# B&R Automation Studio project AAU12Segmenter (part 2)

```iecst
	::OutputVariables[1,0]	AT %QB."KUKA2_KRC4_ProfiNet_5_0".Module001_8_digital_outputs_O_00;
	::OutputVariables[1,1]	AT %QB."KUKA2_KRC4_ProfiNet_5_0".Module001_8_digital_outputs_O_01;
	::OutputVariables[1,2]	AT %QB."KUKA2_KRC4_ProfiNet_5_0".Module001_8_digital_outputs_O_02;
	::OutputVariables[1,3]	AT %QB."KUKA2_KRC4_ProfiNet_5_0".Module001_8_digital_outputs_O_03;
	::OutputVariables[1,4]	AT %QB."KUKA2_KRC4_ProfiNet_5_0".Module001_8_digital_outputs_O_04;
	::OutputVariables[1,5]	AT %QB."KUKA2_KRC4_ProfiNet_5_0".Module001_8_digital_outputs_O_05;
	::OutputVariables[1,6]	AT %QB."KUKA2_KRC4_ProfiNet_5_0".Module001_8_digital_outputs_O_06;
	::OutputVariables[1,7]	AT %QB."KUKA2_KRC4_ProfiNet_5_0".Module001_8_digital_outputs_O_07;
	::OutputVariables[1,8]	AT %QB."KUKA2_KRC4_ProfiNet_5_0".Module001_8_digital_outputs_O_08;
	::OutputVariables[1,9]	AT %QB."KUKA2_KRC4_ProfiNet_5_0".Module001_8_digital_outputs_O_09;
	::OutputVariables[1,10]	AT %QB."KUKA2_KRC4_ProfiNet_5_0".Module001_8_digital_outputs_O_10;
	::OutputVariables[1,11]	AT %QB."KUKA2_KRC4_ProfiNet_5_0".Module001_8_digital_outputs_O_11;
	::OutputVariables[1,12]	AT %QB."KUKA2_KRC4_ProfiNet_5_0".Module001_8_digital_outputs_O_12;
	::OutputVariables[1,13]	AT %QB."KUKA2_KRC4_ProfiNet_5_0".Module001_8_digital_outputs_O_13;
	::OutputVariables[1,14]	AT %QB."KUKA2_KRC4_ProfiNet_5_0".Module001_8_digital_outputs_O_14;
	::OutputVariables[1,15]	AT %QB."KUKA2_KRC4_ProfiNet_5_0".Module001_8_digital_outputs_O_15;
	::OutputVariables[1,16]	AT %QB."KUKA2_KRC4_ProfiNet_5_0".Module001_8_digital_outputs_O_16;
	::OutputVariables[1,17]	AT %QB."KUKA2_KRC4_ProfiNet_5_0".Module001_8_digital_outputs_O_17;
	::OutputVariables[1,18]	AT %QB."KUKA2_KRC4_ProfiNet_5_0".Module001_8_digital_outputs_O_18;
	::OutputVariables[1,19]	AT %QB."KUKA2_KRC4_ProfiNet_5_0".Module001_8_digital_outputs_O_19;
	::OutputVariables[1,20]	AT %QB."KUKA2_KRC4_ProfiNet_5_0".Module001_8_digital_outputs_O_20;
	::OutputVariables[1,21]	AT %QB."KUKA2_KRC4_ProfiNet_5_0".Module001_8_digital_outputs_O_21;
	::OutputVariables[1,22]	AT %QB."KUKA2_KRC4_ProfiNet_5_0".Module001_8_digital_outputs_O_22;
	::OutputVariables[1,23]	AT %QB."KUKA2_KRC4_ProfiNet_5_0".Module001_8_digital_outputs_O_23;
	::OutputVariables[1,24]	AT %QB."KUKA2_KRC4_ProfiNet_5_0".Module001_8_digital_outputs_O_24;
	::OutputVariables[1,25]	AT %QB."KUKA2_KRC4_ProfiNet_5_0".Module001_8_digital_outputs_O_25;
	::OutputVariables[1,26]	AT %QB."KUKA2_KRC4_ProfiNet_5_0".Module001_8_digital_outputs_O_26;
	::OutputVariables[1,27]	AT %QB."KUKA2_KRC4_ProfiNet_5_0".Module001_8_digital_outputs_O_27;
	::OutputVariables[1,28]	AT %QB."KUKA2_KRC4_ProfiNet_5_0".Module001_8_digital_outputs_O_28;
	::OutputVariables[1,29]	AT %QB."KUKA2_KRC4_ProfiNet_5_0".Module001_8_digital_outputs_O_29;
	::OutputVariables[1,30]	AT %QB."KUKA2_KRC4_ProfiNet_5_0".Module001_8_digital_outputs_O_30;
	::OutputVariables[1,31]	AT %QB."KUKA2_KRC4_ProfiNet_5_0".Module001_8_digital_outputs_O_31;
	::OutputVariables[1,32]	AT %QB."KUKA2_KRC4_ProfiNet_5_0".Module001_8_digital_outputs_O_32;
	::OutputVariables[1,33]	AT %QB."KUKA2_KRC4_ProfiNet_5_0".Module001_8_digital_outputs_O_33;
	::OutputVariables[1,34]	AT %QB."KUKA2_KRC4_ProfiNet_5_0".Module001_8_digital_outputs_O_34;
	::OutputVariables[1,35]	AT %QB."KUKA2_KRC4_ProfiNet_5_0".Module001_8_digital_outputs_O_35;
	::OutputVariables[1,36]	AT %QB."KUKA2_KRC4_ProfiNet_5_0".Module001_8_digital_outputs_O_36;
	::OutputVariables[1,37]	AT %QB."KUKA2_KRC4_ProfiNet_5_0".Module001_8_digital_outputs_O_37;
	::OutputVariables[1,38]	AT %QB."KUKA2_KRC4_ProfiNet_5_0".Module001_8_digital_outputs_O_38;
	::OutputVariables[1,39]	AT %QB."KUKA2_KRC4_ProfiNet_5_0".Module001_8_digital_outputs_O_39;
	::OutputVariables[1,40]	AT %QB."KUKA2_KRC4_ProfiNet_5_0".Module001_8_digital_outputs_O_40;
	::OutputVariables[1,41]	AT %QB."KUKA2_KRC4_ProfiNet_5_0".Module001_8_digital_outputs_O_41;
	::OutputVariables[1,42]	AT %QB."KUKA2_KRC4_ProfiNet_5_0".Module001_8_digital_outputs_O_42;
	::OutputVariables[1,43]	AT %QB."KUKA2_KRC4_ProfiNet_5_0".Module001_8_digital_outputs_O_43;
	::OutputVariables[1,44]	AT %QB."KUKA2_KRC4_ProfiNet_5_0".Module001_8_digital_outputs_O_44;
	::OutputVariables[1,45]	AT %QB."KUKA2_KRC4_ProfiNet_5_0".Module001_8_digital_outputs_O_45;
	::OutputVariables[1,46]	AT %QB."KUKA2_KRC4_ProfiNet_5_0".Module001_8_digital_outputs_O_46;
	::OutputVariables[1,47]	AT %QB."KUKA2_KRC4_ProfiNet_5_0".Module001_8_digital_outputs_O_47;
	::OutputVariables[1,48]	AT %QB."KUKA2_KRC4_ProfiNet_5_0".Module001_8_digital_outputs_O_48;
	::OutputVariables[1,49]	AT %QB."KUKA2_KRC4_ProfiNet_5_0".Module001_8_digital_outputs_O_49;
	::OutputVariables[1,50]	AT %QB."KUKA2_KRC4_ProfiNet_5_0".Module001_8_digital_outputs_O_50;
	::OutputVariables[1,51]	AT %QB."KUKA2_KRC4_ProfiNet_5_0".Module001_8_digital_outputs_O_51;
	::OutputVariables[1,52]	AT %QB."KUKA2_KRC4_ProfiNet_5_0".Module001_8_digital_outputs_O_52;
	::OutputVariables[1,53]	AT %QB."KUKA2_KRC4_ProfiNet_5_0".Module001_8_digital_outputs_O_53;
	::OutputVariables[1,54]	AT %QB."KUKA2_KRC4_ProfiNet_5_0".Module001_8_digital_outputs_O_54;
	::OutputVariables[1,55]	AT %QB."KUKA2_KRC4_ProfiNet_5_0".Module001_8_digital_outputs_O_55;
	::OutputVariables[1,56]	AT %QB."KUKA2_KRC4_ProfiNet_5_0".Module001_8_digital_outputs_O_56;
	::OutputVariables[1,57]	AT %QB."KUKA2_KRC4_ProfiNet_5_0".Module001_8_digital_outputs_O_57;
	::OutputVariables[1,58]	AT %QB."KUKA2_KRC4_ProfiNet_5_0".Module001_8_digital_outputs_O_58;
	::OutputVariables[1,59]	AT %QB."KUKA2_KRC4_ProfiNet_5_0".Module001_8_digital_outputs_O_59;
	::OutputVariables[1,60]	AT %QB."KUKA2_KRC4_ProfiNet_5_0".Module001_8_digital_outputs_O_60;
	::OutputVariables[1,61]	AT %QB."KUKA2_KRC4_ProfiNet_5_0".Module001_8_digital_outputs_O_61;
	::OutputVariables[1,62]	AT %QB."KUKA2_KRC4_ProfiNet_5_0".Module001_8_digital_outputs_O_62;
	::OutputVariables[1,63]	AT %QB."KUKA2_KRC4_ProfiNet_5_0".Module001_8_digital_outputs_O_63;
	::OutputVariables[1,64]	AT %QB."KUKA2_KRC4_ProfiNet_5_0".Module001_8_digital_outputs_O_64;
	::OutputVariables[1,65]	AT %QB."KUKA2_KRC4_ProfiNet_5_0".Module001_8_digital_outputs_O_65;
	::OutputVariables[1,66]	AT %QB."KUKA2_KRC4_ProfiNet_5_0".Module001_8_digital_outputs_O_66;
	::OutputVariables[1,67]	AT %QB."KUKA2_KRC4_ProfiNet_5_0".Module001_8_digital_outputs_O_67;
	::OutputVariables[1,68]	AT %QB."KUKA2_KRC4_ProfiNet_5_0".Module001_8_digital_outputs_O_68;
	::OutputVariables[1,69]	AT %QB."KUKA2_KRC4_ProfiNet_5_0".Module001_8_digital_outputs_O_69;
	::OutputVariables[1,70]	AT %QB."KUKA2_KRC4_ProfiNet_5_0".Module001_8_digital_outputs_O_70;
	::OutputVariables[1,71]	AT %QB."KUKA2_KRC4_ProfiNet_5_0".Module001_8_digital_outputs_O_71;
	::OutputVariables[1,72]	AT %QB."KUKA2_KRC4_ProfiNet_5_0".Module001_8_digital_outputs_O_72;
	::OutputVariables[1,73]	AT %QB."KUKA2_KRC4_ProfiNet_5_0".Module001_8_digital_outputs_O_73;
	::OutputVariables[1,74]	AT %QB."KUKA2_KRC4_ProfiNet_5_0".Module001_8_digital_outputs_O_74;
	::OutputVariables[1,75]	AT %QB."KUKA2_KRC4_ProfiNet_5_0".Module001_8_digital_outputs_O_75;
	::OutputVariables[1,76]	AT %QB."KUKA2_KRC4_ProfiNet_5_0".Module001_8_digital_outputs_O_76;
	::OutputVariables[1,77]	AT %QB."KUKA2_KRC4_ProfiNet_5_0".Module001_8_digital_outputs_O_77;
	::OutputVariables[1,78]	AT %QB."KUKA2_KRC4_ProfiNet_5_0".Module001_8_digital_outputs_O_78;
	::OutputVariables[1,79]	AT %QB."KUKA2_KRC4_ProfiNet_5_0".Module001_8_digital_outputs_O_79;
	::OutputVariables[1,80]	AT %QB."KUKA2_KRC4_ProfiNet_5_0".Module001_8_digital_outputs_O_80;
	::OutputVariables[1,81]	AT %QB."KUKA2_KRC4_ProfiNet_5_0".Module001_8_digital_outputs_O_81;
	::OutputVariables[1,82]	AT %QB."KUKA2_KRC4_ProfiNet_5_0".Module001_8_digital_outputs_O_82;
	::OutputVariables[1,83]	AT %QB."KUKA2_KRC4_ProfiNet_5_0".Module001_8_digital_outputs_O_83;
	::OutputVariables[1,84]	AT %QB."KUKA2_KRC4_ProfiNet_5_0".Module001_8_digital_outputs_O_84;
	::OutputVariables[1,85]	AT %QB."KUKA2_KRC4_ProfiNet_5_0".Module001_8_digital_outputs_O_85;
	::OutputVariables[1,86]	AT %QB."KUKA2_KRC4_ProfiNet_5_0".Module001_8_digital_outputs_O_86;
	::OutputVariables[1,87]	AT %QB."KUKA2_KRC4_ProfiNet_5_0".Module001_8_digital_outputs_O_87;
	::OutputVariables[1,88]	AT %QB."KUKA2_KRC4_ProfiNet_5_0".Module001_8_digital_outputs_O_88;
	::OutputVariables[1,89]	AT %QB."KUKA2_KRC4_ProfiNet_5_0".Module001_8_digital_outputs_O_89;
	::OutputVariables[1,90]	AT %QB."KUKA2_KRC4_ProfiNet_5_0".Module001_8_digital_outputs_O_90;
	::OutputVariables[1,91]	AT %QB."KUKA2_KRC4_ProfiNet_5_0".Module001_8_digital_outputs_O_91;
	::OutputVariables[1,92]	AT %QB."KUKA2_KRC4_ProfiNet_5_0".Module001_8_digital_outputs_O_92;
	::OutputVariables[1,93]	AT %QB."KUKA2_KRC4_ProfiNet_5_0".Module001_8_digital_outputs_O_93;
	::OutputVariables[1,94]	AT %QB."KUKA2_KRC4_ProfiNet_5_0".Module001_8_digital_outputs_O_94;
	::OutputVariables[1,95]	AT %QB."KUKA2_KRC4_ProfiNet_5_0".Module001_8_digital_outputs_O_95;
	::OutputVariables[1,96]	AT %QB."KUKA2_KRC4_ProfiNet_5_0".Module001_8_digital_outputs_O_96;
	::OutputVariables[1,97]	AT %QB."KUKA2_KRC4_ProfiNet_5_0".Module001_8_digital_outputs_O_97;
	::OutputVariables[1,98]	AT %QB."KUKA2_KRC4_ProfiNet_5_0".Module001_8_digital_outputs_O_98;
	::OutputVariables[1,99]	AT %QB."KUKA2_KRC4_ProfiNet_5_0".Module001_8_digital_outputs_O_99;
	::OutputVariables[1,100]	AT %QB."KUKA2_KRC4_ProfiNet_5_0".Module001_8_digital_outputs_O_100;
	::OutputVariables[1,101]	AT %QB."KUKA2_KRC4_ProfiNet_5_0".Module001_8_digital_outputs_O_101;
	::OutputVariables[1,102]	AT %QB."KUKA2_KRC4_ProfiNet_5_0".Module001_8_digital_outputs_O_102;
	::OutputVariables[1,103]	AT %QB."KUKA2_KRC4_ProfiNet_5_0".Module001_8_digital_outputs_O_103;
	::OutputVariables[1,104]	AT %QB."KUKA2_KRC4_ProfiNet_5_0".Module001_8_digital_outputs_O_104;
	::OutputVariables[1,105]	AT %QB."KUKA2_KRC4_ProfiNet_5_0".Module001_8_digital_outputs_O_105;
	::OutputVariables[1,106]	AT %QB."KUKA2_KRC4_ProfiNet_5_0".Module001_8_digital_outputs_O_106;
	::OutputVariables[1,107]	AT %QB."KUKA2_KRC4_ProfiNet_5_0".Module001_8_digital_outputs_O_107;
	::OutputVariables[1,108]	AT %QB."KUKA2_KRC4_ProfiNet_5_0".Module001_8_digital_outputs_O_108;
	::OutputVariables[1,109]	AT %QB."KUKA2_KRC4_ProfiNet_5_0".Module001_8_digital_outputs_O_109;
	::OutputVariables[1,110]	AT %QB."KUKA2_KRC4_ProfiNet_5_0".Module001_8_digital_outputs_O_110;
	::OutputVariables[1,111]	AT %QB."KUKA2_KRC4_ProfiNet_5_0".Module001_8_digital_outputs_O_111;
	::OutputVariables[1,112]	AT %QB."KUKA2_KRC4_ProfiNet_5_0".Module001_8_digital_outputs_O_112;
	::OutputVariables[1,113]	AT %QB."KUKA2_KRC4_ProfiNet_5_0".Module001_8_digital_outputs_O_113;
	::OutputVariables[1,114]	AT %QB."KUKA2_KRC4_ProfiNet_5_0".Module001_8_digital_outputs_O_114;
	::OutputVariables[1,115]	AT %QB."KUKA2_KRC4_ProfiNet_5_0".Module001_8_digital_outputs_O_115;
	::OutputVariables[1,116]	AT %QB."KUKA2_KRC4_ProfiNet_5_0".Module001_8_digital_outputs_O_116;
	::OutputVariables[1,117]	AT %QB."KUKA2_KRC4_ProfiNet_5_0".Module001_8_digital_outputs_O_117;
	::OutputVariables[1,118]	AT %QB."KUKA2_KRC4_ProfiNet_5_0".Module001_8_digital_outputs_O_118;
	::OutputVariables[1,119]	AT %QB."KUKA2_KRC4_ProfiNet_5_0".Module001_8_digital_outputs_O_119;
	::OutputVariables[1,120]	AT %QB."KUKA2_KRC4_ProfiNet_5_0".Module001_8_digital_outputs_O_120;
	::OutputVariables[1,121]	AT %QB."KUKA2_KRC4_ProfiNet_5_0".Module001_8_digital_outputs_O_121;
	::OutputVariables[1,122]	AT %QB."KUKA2_KRC4_ProfiNet_5_0".Module001_8_digital_outputs_O_122;
	::OutputVariables[1,123]	AT %QB."KUKA2_KRC4_ProfiNet_5_0".Module001_8_digital_outputs_O_123;
	::OutputVariables[1,124]	AT %QB."KUKA2_KRC4_ProfiNet_5_0".Module001_8_digital_outputs_O_124;
	::OutputVariables[1,125]	AT %QB."KUKA2_KRC4_ProfiNet_5_0".Module001_8_digital_outputs_O_125;
	::OutputVariables[1,126]	AT %QB."KUKA2_KRC4_ProfiNet_5_0".Module001_8_digital_outputs_O_126;
	::OutputVariables[1,127]	AT %QB."KUKA2_KRC4_ProfiNet_5_0".Module001_8_digital_outputs_O_127;
	::OutputVariables[1,128]	AT %QB."KUKA2_KRC4_ProfiNet_5_0".Module001_8_digital_outputs_O_128;
	::OutputVariables[1,129]	AT %QB."KUKA2_KRC4_ProfiNet_5_0".Module001_8_digital_outputs_O_129;
	::OutputVariables[1,130]	AT %QB."KUKA2_KRC4_ProfiNet_5_0".Module001_8_digital_outputs_O_130;
	::OutputVariables[1,131]	AT %QB."KUKA2_KRC4_ProfiNet_5_0".Module001_8_digital_outputs_O_131;
	::OutputVariables[1,132]	AT %QB."KUKA2_KRC4_ProfiNet_5_0".Module001_8_digital_outputs_O_132;
	::OutputVariables[1,133]	AT %QB."KUKA2_KRC4_ProfiNet_5_0".Module001_8_digital_outputs_O_133;
	::OutputVariables[1,134]	AT %QB."KUKA2_KRC4_ProfiNet_5_0".Module001_8_digital_outputs_O_134;
	::OutputVariables[1,135]	AT %QB."KUKA2_KRC4_ProfiNet_5_0".Module001_8_digital_outputs_O_135;
	::OutputVariables[1,136]	AT %QB."KUKA2_KRC4_ProfiNet_5_0".Module001_8_digital_outputs_O_136;
	::OutputVariables[1,137]	AT %QB."KUKA2_KRC4_ProfiNet_5_0".Module001_8_digital_outputs_O_137;
	::OutputVariables[1,138]	AT %QB."KUKA2_KRC4_ProfiNet_5_0".Module001_8_digital_outputs_O_138;
	::OutputVariables[1,139]	AT %QB."KUKA2_KRC4_ProfiNet_5_0".Module001_8_digital_outputs_O_139;
	::OutputVariables[1,140]	AT %QB."KUKA2_KRC4_ProfiNet_5_0".Module001_8_digital_outputs_O_140;
	::OutputVariables[1,141]	AT %QB."KUKA2_KRC4_ProfiNet_5_0".Module001_8_digital_outputs_O_141;
	::OutputVariables[1,142]	AT %QB."KUKA2_KRC4_ProfiNet_5_0".Module001_8_digital_outputs_O_142;
	::OutputVariables[1,143]	AT %QB."KUKA2_KRC4_ProfiNet_5_0".Module001_8_digital_outputs_O_143;
	::OutputVariables[1,144]	AT %QB."KUKA2_KRC4_ProfiNet_5_0".Module001_8_digital_outputs_O_144;
	::OutputVariables[1,145]	AT %QB."KUKA2_KRC4_ProfiNet_5_0".Module001_8_digital_outputs_O_145;
	::OutputVariables[1,146]	AT %QB."KUKA2_KRC4_ProfiNet_5_0".Module001_8_digital_outputs_O_146;
	::OutputVariables[1,147]	AT %QB."KUKA2_KRC4_ProfiNet_5_0".Module001_8_digital_outputs_O_147;
	::OutputVariables[1,148]	AT %QB."KUKA2_KRC4_ProfiNet_5_0".Module001_8_digital_outputs_O_148;
	::OutputVariables[1,149]	AT %QB."KUKA2_KRC4_ProfiNet_5_0".Module001_8_digital_outputs_O_149;
	::OutputVariables[1,150]	AT %QB."KUKA2_KRC4_ProfiNet_5_0".Module001_8_digital_outputs_O_150;
	::OutputVariables[1,151]	AT %QB."KUKA2_KRC4_ProfiNet_5_0".Module001_8_digital_outputs_O_151;
	::OutputVariables[1,152]	AT %QB."KUKA2_KRC4_ProfiNet_5_0".Module001_8_digital_outputs_O_152;
	::OutputVariables[1,153]	AT %QB."KUKA2_KRC4_ProfiNet_5_0".Module001_8_digital_outputs_O_153;
	::OutputVariables[1,154]	AT %QB."KUKA2_KRC4_ProfiNet_5_0".Module001_8_digital_outputs_O_154;
	::OutputVariables[1,155]	AT %QB."KUKA2_KRC4_ProfiNet_5_0".Module001_8_digital_outputs_O_155;
	::OutputVariables[1,156]	AT %QB."KUKA2_KRC4_ProfiNet_5_0".Module001_8_digital_outputs_O_156;
	::OutputVariables[1,157]	AT %QB."KUKA2_KRC4_ProfiNet_5_0".Module001_8_digital_outputs_O_157;
	::OutputVariables[1,158]	AT %QB."KUKA2_KRC4_ProfiNet_5_0".Module001_8_digital_outputs_O_158;
	::OutputVariables[1,159]	AT %QB."KUKA2_KRC4_ProfiNet_5_0".Module001_8_digital_outputs_O_159;
	::OutputVariables[1,160]	AT %QB."KUKA2_KRC4_ProfiNet_5_0".Module001_8_digital_outputs_O_160;
	::OutputVariables[1,161]	AT %QB."KUKA2_KRC4_ProfiNet_5_0".Module001_8_digital_outputs_O_161;
	::OutputVariables[1,162]	AT %QB."KUKA2_KRC4_ProfiNet_5_0".Module001_8_digital_outputs_O_162;
	::OutputVariables[1,163]	AT %QB."KUKA2_KRC4_ProfiNet_5_0".Module001_8_digital_outputs_O_163;
	::OutputVariables[1,164]	AT %QB."KUKA2_KRC4_ProfiNet_5_0".Module001_8_digital_outputs_O_164;
	::OutputVariables[1,165]	AT %QB."KUKA2_KRC4_ProfiNet_5_0".Module001_8_digital_outputs_O_165;
	::OutputVariables[1,166]	AT %QB."KUKA2_KRC4_ProfiNet_5_0".Module001_8_digital_outputs_O_166;
	::OutputVariables[1,167]	AT %QB."KUKA2_KRC4_ProfiNet_5_0".Module001_8_digital_outputs_O_167;
	::OutputVariables[1,168]	AT %QB."KUKA2_KRC4_ProfiNet_5_0".Module001_8_digital_outputs_O_168;
	::OutputVariables[1,169]	AT %QB."KUKA2_KRC4_ProfiNet_5_0".Module001_8_digital_outputs_O_169;
	::OutputVariables[1,170]	AT %QB."KUKA2_KRC4_ProfiNet_5_0".Module001_8_digital_outputs_O_170;
	::OutputVariables[1,171]	AT %QB."KUKA2_KRC4_ProfiNet_5_0".Module001_8_digital_outputs_O_171;
	::OutputVariables[1,172]	AT %QB."KUKA2_KRC4_ProfiNet_5_0".Module001_8_digital_outputs_O_172;
	::OutputVariables[1,173]	AT %QB."KUKA2_KRC4_ProfiNet_5_0".Module001_8_digital_outputs_O_173;
	::OutputVariables[1,174]	AT %QB."KUKA2_KRC4_ProfiNet_5_0".Module001_8_digital_outputs_O_174;
	::OutputVariables[1,175]	AT %QB."KUKA2_KRC4_ProfiNet_5_0".Module001_8_digital_outputs_O_175;
	::OutputVariables[1,176]	AT %QB."KUKA2_KRC4_ProfiNet_5_0".Module001_8_digital_outputs_O_176;
	::OutputVariables[1,177]	AT %QB."KUKA2_KRC4_ProfiNet_5_0".Module001_8_digital_outputs_O_177;
	::OutputVariables[1,178]	AT %QB."KUKA2_KRC4_ProfiNet_5_0".Module001_8_digital_outputs_O_178;
	::OutputVariables[1,179]	AT %QB."KUKA2_KRC4_ProfiNet_5_0".Module001_8_digital_outputs_O_179;
	::OutputVariables[1,180]	AT %QB."KUKA2_KRC4_ProfiNet_5_0".Module001_8_digital_outputs_O_180;
	::OutputVariables[1,181]	AT %QB."KUKA2_KRC4_ProfiNet_5_0".Module001_8_digital_outputs_O_181;
	::OutputVariables[1,182]	AT %QB."KUKA2_KRC4_ProfiNet_5_0".Module001_8_digital_outputs_O_182;
	::OutputVariables[1,183]	AT %QB."KUKA2_KRC4_ProfiNet_5_0".Module001_8_digital_outputs_O_183;
	::OutputVariables[1,184]	AT %QB."KUKA2_KRC4_ProfiNet_5_0".Module001_8_digital_outputs_O_184;
	::OutputVariables[1,185]	AT %QB."KUKA2_KRC4_ProfiNet_5_0".Module001_8_digital_outputs_O_185;
	::OutputVariables[1,186]	AT %QB."KUKA2_KRC4_ProfiNet_5_0".Module001_8_digital_outputs_O_186;
	::OutputVariables[1,187]	AT %QB."KUKA2_KRC4_ProfiNet_5_0".Module001_8_digital_outputs_O_187;
	::OutputVariables[1,188]	AT %QB."KUKA2_KRC4_ProfiNet_5_0".Module001_8_digital_outputs_O_188;
	::OutputVariables[1,189]	AT %QB."KUKA2_KRC4_ProfiNet_5_0".Module001_8_digital_outputs_O_189;
	::OutputVariables[1,190]	AT %QB."KUKA2_KRC4_ProfiNet_5_0".Module001_8_digital_outputs_O_190;
	::OutputVariables[1,191]	AT %QB."KUKA2_KRC4_ProfiNet_5_0".Module001_8_digital_outputs_O_191;
	::OutputVariables[1,192]	AT %QB."KUKA2_KRC4_ProfiNet_5_0".Module001_8_digital_outputs_O_192;
	::OutputVariables[1,193]	AT %QB."KUKA2_KRC4_ProfiNet_5_0".Module001_8_digital_outputs_O_193;
	::OutputVariables[1,194]	AT %QB."KUKA2_KRC4_ProfiNet_5_0".Module001_8_digital_outputs_O_194;
	::OutputVariables[1,195]	AT %QB."KUKA2_KRC4_ProfiNet_5_0".Module001_8_digital_outputs_O_195;
	::OutputVariables[1,196]	AT %QB."KUKA2_KRC4_ProfiNet_5_0".Module001_8_digital_outputs_O_196;
	::OutputVariables[1,197]	AT %QB."KUKA2_KRC4_ProfiNet_5_0".Module001_8_digital_outputs_O_197;
	::OutputVariables[1,198]	AT %QB."KUKA2_KRC4_ProfiNet_5_0".Module001_8_digital_outputs_O_198;
	::OutputVariables[1,199]	AT %QB."KUKA2_KRC4_ProfiNet_5_0".Module001_8_digital_outputs_O_199;
	::OutputVariables[1,200]	AT %QB."KUKA2_KRC4_ProfiNet_5_0".Module001_8_digital_outputs_O_200;
	::OutputVariables[1,201]	AT %QB."KUKA2_KRC4_ProfiNet_5_0".Module001_8_digital_outputs_O_201;
	::OutputVariables[1,202]	AT %QB."KUKA2_KRC4_ProfiNet_5_0".Module001_8_digital_outputs_O_202;
	::OutputVariables[1,203]	AT %QB."KUKA2_KRC4_ProfiNet_5_0".Module001_8_digital_outputs_O_203;
	::OutputVariables[1,204]	AT %QB."KUKA2_KRC4_ProfiNet_5_0".Module001_8_digital_outputs_O_204;
	::OutputVariables[1,205]	AT %QB."KUKA2_KRC4_ProfiNet_5_0".Module001_8_digital_outputs_O_205;
	::OutputVariables[1,206]	AT %QB."KUKA2_KRC4_ProfiNet_5_0".Module001_8_digital_outputs_O_206;
	::OutputVariables[1,207]	AT %QB."KUKA2_KRC4_ProfiNet_5_0".Module001_8_digital_outputs_O_207;
	::OutputVariables[1,208]	AT %QB."KUKA2_KRC4_ProfiNet_5_0".Module001_8_digital_outputs_O_208;
	::OutputVariables[1,209]	AT %QB."KUKA2_KRC4_ProfiNet_5_0".Module001_8_digital_outputs_O_209;
	::OutputVariables[1,210]	AT %QB."KUKA2_KRC4_ProfiNet_5_0".Module001_8_digital_outputs_O_210;
	::OutputVariables[1,211]	AT %QB."KUKA2_KRC4_ProfiNet_5_0".Module001_8_digital_outputs_O_211;
	::OutputVariables[1,212]	AT %QB."KUKA2_KRC4_ProfiNet_5_0".Module001_8_digital_outputs_O_212;
	::OutputVariables[1,213]	AT %QB."KUKA2_KRC4_ProfiNet_5_0".Module001_8_digital_outputs_O_213;
	::OutputVariables[1,214]	AT %QB."KUKA2_KRC4_ProfiNet_5_0".Module001_8_digital_outputs_O_214;
	::OutputVariables[1,215]	AT %QB."KUKA2_KRC4_ProfiNet_5_0".Module001_8_digital_outputs_O_215;
	::OutputVariables[1,216]	AT %QB."KUKA2_KRC4_ProfiNet_5_0".Module001_8_digital_outputs_O_216;
	::OutputVariables[1,217]	AT %QB."KUKA2_KRC4_ProfiNet_5_0".Module001_8_digital_outputs_O_217;
	::OutputVariables[1,218]	AT %QB."KUKA2_KRC4_ProfiNet_5_0".Module001_8_digital_outputs_O_218;
	::OutputVariables[1,219]	AT %QB."KUKA2_KRC4_ProfiNet_5_0".Module001_8_digital_outputs_O_219;
	::OutputVariables[1,220]	AT %QB."KUKA2_KRC4_ProfiNet_5_0".Module001_8_digital_outputs_O_220;
	::OutputVariables[1,221]	AT %QB."KUKA2_KRC4_ProfiNet_5_0".Module001_8_digital_outputs_O_221;
	::OutputVariables[1,222]	AT %QB."KUKA2_KRC4_ProfiNet_5_0".Module001_8_digital_outputs_O_222;
	::OutputVariables[1,223]	AT %QB."KUKA2_KRC4_ProfiNet_5_0".Module001_8_digital_outputs_O_223;
	::OutputVariables[1,224]	AT %QB."KUKA2_KRC4_ProfiNet_5_0".Module001_8_digital_outputs_O_224;
	::OutputVariables[1,225]	AT %QB."KUKA2_KRC4_ProfiNet_5_0".Module001_8_digital_outputs_O_225;
	::OutputVariables[1,226]	AT %QB."KUKA2_KRC4_ProfiNet_5_0".Module001_8_digital_outputs_O_226;
	::OutputVariables[1,227]	AT %QB."KUKA2_KRC4_ProfiNet_5_0".Module001_8_digital_outputs_O_227;
	::OutputVariables[1,228]	AT %QB."KUKA2_KRC4_ProfiNet_5_0".Module001_8_digital_outputs_O_228;
	::OutputVariables[1,229]	AT %QB."KUKA2_KRC4_ProfiNet_5_0".Module001_8_digital_outputs_O_229;
	::OutputVariables[1,230]	AT %QB."KUKA2_KRC4_ProfiNet_5_0".Module001_8_digital_outputs_O_230;
	::OutputVariables[1,231]	AT %QB."KUKA2_KRC4_ProfiNet_5_0".Module001_8_digital_outputs_O_231;
	::OutputVariables[1,232]	AT %QB."KUKA2_KRC4_ProfiNet_5_0".Module001_8_digital_outputs_O_232;
	::OutputVariables[1,233]	AT %QB."KUKA2_KRC4_ProfiNet_5_0".Module001_8_digital_outputs_O_233;
	::OutputVariables[1,234]	AT %QB."KUKA2_KRC4_ProfiNet_5_0".Module001_8_digital_outputs_O_234;
	::OutputVariables[1,235]	AT %QB."KUKA2_KRC4_ProfiNet_5_0".Module001_8_digital_outputs_O_235;
	::OutputVariables[1,236]	AT %QB."KUKA2_KRC4_ProfiNet_5_0".Module001_8_digital_outputs_O_236;
	::OutputVariables[1,237]	AT %QB."KUKA2_KRC4_ProfiNet_5_0".Module001_8_digital_outputs_O_237;
	::OutputVariables[1,238]	AT %QB."KUKA2_KRC4_ProfiNet_5_0".Module001_8_digital_outputs_O_238;
	::OutputVariables[1,239]	AT %QB."KUKA2_KRC4_ProfiNet_5_0".Module001_8_digital_outputs_O_239;
	::OutputVariables[1,240]	AT %QB."KUKA2_KRC4_ProfiNet_5_0".Module001_8_digital_outputs_O_240;
	::OutputVariables[1,241]	AT %QB."KUKA2_KRC4_ProfiNet_5_0".Module001_8_digital_outputs_O_241;
	::OutputVariables[1,242]	AT %QB."KUKA2_KRC4_ProfiNet_5_0".Module001_8_digital_outputs_O_242;
	::OutputVariables[1,243]	AT %QB."KUKA2_KRC4_ProfiNet_5_0".Module001_8_digital_outputs_O_243;
	::OutputVariables[1,244]	AT %QB."KUKA2_KRC4_ProfiNet_5_0".Module001_8_digital_outputs_O_244;
	::OutputVariables[1,245]	AT %QB."KUKA2_KRC4_ProfiNet_5_0".Module001_8_digital_outputs_O_245;
	::OutputVariables[1,246]	AT %QB."KUKA2_KRC4_ProfiNet_5_0".Module001_8_digital_outputs_O_246;
	::OutputVariables[1,247]	AT %QB."KUKA2_KRC4_ProfiNet_5_0".Module001_8_digital_outputs_O_247;
	::OutputVariables[1,248]	AT %QB."KUKA2_KRC4_ProfiNet_5_0".Module001_8_digital_outputs_O_248;
	::OutputVariables[1,249]	AT %QB."KUKA2_KRC4_ProfiNet_5_0".Module001_8_digital_outputs_O_249;
	::OutputVariables[1,250]	AT %QB."KUKA2_KRC4_ProfiNet_5_0".Module001_8_digital_outputs_O_250;
	::OutputVariables[1,251]	AT %QB."KUKA2_KRC4_ProfiNet_5_0".Module001_8_digital_outputs_O_251;
	::OutputVariables[1,252]	AT %QB."KUKA2_KRC4_ProfiNet_5_0".Module001_8_digital_outputs_O_252;
	::OutputVariables[1,253]	AT %QB."KUKA2_KRC4_ProfiNet_5_0".Module001_8_digital_outputs_O_253;

	(*________________________________________*)
	(*_____________KUKA3 Mappings_____________*)
	(*________________________________________*)

	::InputVariables[2,0] AT %IB."KUKA3_KRC4_ProfiNet_5_0".Module001_8_digital_inputs_I_00;
	::InputVariables[2,1] AT %IB."KUKA3_KRC4_ProfiNet_5_0".Module001_8_digital_inputs_I_01;
	::InputVariables[2,2] AT %IB."KUKA3_KRC4_ProfiNet_5_0".Module001_8_digital_inputs_I_02;
	::InputVariables[2,3] AT %IB."KUKA3_KRC4_ProfiNet_5_0".Module001_8_digital_inputs_I_03;
	::InputVariables[2,4] AT %IB."KUKA3_KRC4_ProfiNet_5_0".Module001_8_digital_inputs_I_04;
	::InputVariables[2,5] AT %IB."KUKA3_KRC4_ProfiNet_5_0".Module001_8_digital_inputs_I_05;
	::InputVariables[2,6] AT %IB."KUKA3_KRC4_ProfiNet_5_0".Module001_8_digital_inputs_I_06;
	::InputVariables[2,7] AT %IB."KUKA3_KRC4_ProfiNet_5_0".Module001_8_digital_inputs_I_07;
	::InputVariables[2,8] AT %IB."KUKA3_KRC4_ProfiNet_5_0".Module001_8_digital_inputs_I_08;
	::InputVariables[2,9] AT %IB."KUKA3_KRC4_ProfiNet_5_0".Module001_8_digital_inputs_I_09;
	::InputVariables[2,10] AT %IB."KUKA3_KRC4_ProfiNet_5_0".Module001_8_digital_inputs_I_10;
	::InputVariables[2,11] AT %IB."KUKA3_KRC4_ProfiNet_5_0".Module001_8_digital_inputs_I_11;
	::InputVariables[2,12] AT %IB."KUKA3_KRC4_ProfiNet_5_0".Module001_8_digital_inputs_I_12;
	::InputVariables[2,13] AT %IB."KUKA3_KRC4_ProfiNet_5_0".Module001_8_digital_inputs_I_13;
	::InputVariables[2,14] AT %IB."KUKA3_KRC4_ProfiNet_5_0".Module001_8_digital_inputs_I_14;
	::InputVariables[2,15] AT %IB."KUKA3_KRC4_ProfiNet_5_0".Module001_8_digital_inputs_I_15;
	::InputVariables[2,16] AT %IB."KUKA3_KRC4_ProfiNet_5_0".Module001_8_digital_inputs_I_16;
	::InputVariables[2,17] AT %IB."KUKA3_KRC4_ProfiNet_5_0".Module001_8_digital_inputs_I_17;
	::InputVariables[2,18] AT %IB."KUKA3_KRC4_ProfiNet_5_0".Module001_8_digital_inputs_I_18;
	::InputVariables[2,19] AT %IB."KUKA3_KRC4_ProfiNet_5_0".Module001_8_digital_inputs_I_19;
	::InputVariables[2,20] AT %IB."KUKA3_KRC4_ProfiNet_5_0".Module001_8_digital_inputs_I_20;
	::InputVariables[2,21] AT %IB."KUKA3_KRC4_ProfiNet_5_0".Module001_8_digital_inputs_I_21;
	::InputVariables[2,22] AT %IB."KUKA3_KRC4_ProfiNet_5_0".Module001_8_digital_inputs_I_22;
	::InputVariables[2,23] AT %IB."KUKA3_KRC4_ProfiNet_5_0".Module001_8_digital_inputs_I_23;
	::InputVariables[2,24] AT %IB."KUKA3_KRC4_ProfiNet_5_0".Module001_8_digital_inputs_I_24;
	::InputVariables[2,25] AT %IB."KUKA3_KRC4_ProfiNet_5_0".Module001_8_digital_inputs_I_25;
	::InputVariables[2,26] AT %IB."KUKA3_KRC4_ProfiNet_5_0".Module001_8_digital_inputs_I_26;
	::InputVariables[2,27] AT %IB."KUKA3_KRC4_ProfiNet_5_0".Module001_8_digital_inputs_I_27;
	::InputVariables[2,28] AT %IB."KUKA3_KRC4_ProfiNet_5_0".Module001_8_digital_inputs_I_28;
	::InputVariables[2,29] AT %IB."KUKA3_KRC4_ProfiNet_5_0".Module001_8_digital_inputs_I_29;
	::InputVariables[2,30] AT %IB."KUKA3_KRC4_ProfiNet_5_0".Module001_8_digital_inputs_I_30;
	::InputVariables[2,31] AT %IB."KUKA3_KRC4_ProfiNet_5_0".Module001_8_digital_inputs_I_31;
	::InputVariables[2,32] AT %IB."KUKA3_KRC4_ProfiNet_5_0".Module001_8_digital_inputs_I_32;
	::InputVariables[2,33] AT %IB."KUKA3_KRC4_ProfiNet_5_0".Module001_8_digital_inputs_I_33;
	::InputVariables[2,34] AT %IB."KUKA3_KRC4_ProfiNet_5_0".Module001_8_digital_inputs_I_34;
	::InputVariables[2,35] AT %IB."KUKA3_KRC4_ProfiNet_5_0".Module001_8_digital_inputs_I_35;
	::InputVariables[2,36] AT %IB."KUKA3_KRC4_ProfiNet_5_0".Module001_8_digital_inputs_I_36;
	::InputVariables[2,37] AT %IB."KUKA3_KRC4_ProfiNet_5_0".Module001_8_digital_inputs_I_37;
	::InputVariables[2,38] AT %IB."KUKA3_KRC4_ProfiNet_5_0".Module001_8_digital_inputs_I_38;
	::InputVariables[2,39] AT %IB."KUKA3_KRC4_ProfiNet_5_0".Module001_8_digital_inputs_I_39;
	::InputVariables[2,40] AT %IB."KUKA3_KRC4_ProfiNet_5_0".Module001_8_digital_inputs_I_40;
	::InputVariables[2,41] AT %IB."KUKA3_KRC4_ProfiNet_5_0".Module001_8_digital_inputs_I_41;
	::InputVariables[2,42] AT %IB."KUKA3_KRC4_ProfiNet_5_0".Module001_8_digital_inputs_I_42;
	::InputVariables[2,43] AT %IB."KUKA3_KRC4_ProfiNet_5_0".Module001_8_digital_inputs_I_43;
	::InputVariables[2,44] AT %IB."KUKA3_KRC4_ProfiNet_5_0".Module001_8_digital_inputs_I_44;
	::InputVariables[2,45] AT %IB."KUKA3_KRC4_ProfiNet_5_0".Module001_8_digital_inputs_I_45;
	::InputVariables[2,46] AT %IB."KUKA3_KRC4_ProfiNet_5_0".Module001_8_digital_inputs_I_46;
	::InputVariables[2,47] AT %IB."KUKA3_KRC4_ProfiNet_5_0".Module001_8_digital_inputs_I_47;
	::InputVariables[2,48] AT %IB."KUKA3_KRC4_ProfiNet_5_0".Module001_8_digital_inputs_I_48;
	::InputVariables[2,49] AT %IB."KUKA3_KRC4_ProfiNet_5_0".Module001_8_digital_inputs_I_49;
	::InputVariables[2,50] AT %IB."KUKA3_KRC4_ProfiNet_5_0".Module001_8_digital_inputs_I_50;
	::InputVariables[2,51] AT %IB."KUKA3_KRC4_ProfiNet_5_0".Module001_8_digital_inputs_I_51;
	::InputVariables[2,52] AT %IB."KUKA3_KRC4_ProfiNet_5_0".Module001_8_digital_inputs_I_52;
	::InputVariables[2,53] AT %IB."KUKA3_KRC4_ProfiNet_5_0".Module001_8_digital_inputs_I_53;
	::InputVariables[2,54] AT %IB."KUKA3_KRC4_ProfiNet_5_0".Module001_8_digital_inputs_I_54;
	::InputVariables[2,55] AT %IB."KUKA3_KRC4_ProfiNet_5_0".Module001_8_digital_inputs_I_55;
	::InputVariables[2,56] AT %IB."KUKA3_KRC4_ProfiNet_5_0".Module001_8_digital_inputs_I_56;
	::InputVariables[2,57] AT %IB."KUKA3_KRC4_ProfiNet_5_0".Module001_8_digital_inputs_I_57;
	::InputVariables[2,58] AT %IB."KUKA3_KRC4_ProfiNet_5_0".Module001_8_digital_inputs_I_58;
	::InputVariables[2,59] AT %IB."KUKA3_KRC4_ProfiNet_5_0".Module001_8_digital_inputs_I_59;
	::InputVariables[2,60] AT %IB."KUKA3_KRC4_ProfiNet_5_0".Module001_8_digital_inputs_I_60;
	::InputVariables[2,61] AT %IB."KUKA3_KRC4_ProfiNet_5_0".Module001_8_digital_inputs_I_61;
	::InputVariables[2,62] AT %IB."KUKA3_KRC4_ProfiNet_5_0".Module001_8_digital_inputs_I_62;
	::InputVariables[2,63] AT %IB."KUKA3_KRC4_ProfiNet_5_0".Module001_8_digital_inputs_I_63;
	::InputVariables[2,64] AT %IB."KUKA3_KRC4_ProfiNet_5_0".Module001_8_digital_inputs_I_64;
	::InputVariables[2,65] AT %IB."KUKA3_KRC4_ProfiNet_5_0".Module001_8_digital_inputs_I_65;
	::InputVariables[2,66] AT %IB."KUKA3_KRC4_ProfiNet_5_0".Module001_8_digital_inputs_I_66;
	::InputVariables[2,67] AT %IB."KUKA3_KRC4_ProfiNet_5_0".Module001_8_digital_inputs_I_67;
	::InputVariables[2,68] AT %IB."KUKA3_KRC4_ProfiNet_5_0".Module001_8_digital_inputs_I_68;
	::InputVariables[2,69] AT %IB."KUKA3_KRC4_ProfiNet_5_0".Module001_8_digital_inputs_I_69;
	::InputVariables[2,70] AT %IB."KUKA3_KRC4_ProfiNet_5_0".Module001_8_digital_inputs_I_70;
	::InputVariables[2,71] AT %IB."KUKA3_KRC4_ProfiNet_5_0".Module001_8_digital_inputs_I_71;
	::InputVariables[2,72] AT %IB."KUKA3_KRC4_ProfiNet_5_0".Module001_8_digital_inputs_I_72;
	::InputVariables[2,73] AT %IB."KUKA3_KRC4_ProfiNet_5_0".Module001_8_digital_inputs_I_73;
	::InputVariables[2,74] AT %IB."KUKA3_KRC4_ProfiNet_5_0".Module001_8_digital_inputs_I_74;
	::InputVariables[2,75] AT %IB."KUKA3_KRC4_ProfiNet_5_0".Module001_8_digital_inputs_I_75;
	::InputVariables[2,76] AT %IB."KUKA3_KRC4_ProfiNet_5_0".Module001_8_digital_inputs_I_76;
	::InputVariables[2,77] AT %IB."KUKA3_KRC4_ProfiNet_5_0".Module001_8_digital_inputs_I_77;
	::InputVariables[2,78] AT %IB."KUKA3_KRC4_ProfiNet_5_0".Module001_8_digital_inputs_I_78;
	::InputVariables[2,79] AT %IB."KUKA3_KRC4_ProfiNet_5_0".Module001_8_digital_inputs_I_79;
	::InputVariables[2,80] AT %IB."KUKA3_KRC4_ProfiNet_5_0".Module001_8_digital_inputs_I_80;
	::InputVariables[2,81] AT %IB."KUKA3_KRC4_ProfiNet_5_0".Module001_8_digital_inputs_I_81;
	::InputVariables[2,82] AT %IB."KUKA3_KRC4_ProfiNet_5_0".Module001_8_digital_inputs_I_82;
	::InputVariables[2,83] AT %IB."KUKA3_KRC4_ProfiNet_5_0".Module001_8_digital_inputs_I_83;
	::InputVariables[2,84] AT %IB."KUKA3_KRC4_ProfiNet_5_0".Module001_8_digital_inputs_I_84;
	::InputVariables[2,85] AT %IB."KUKA3_KRC4_ProfiNet_5_0".Module001_8_digital_inputs_I_85;
	::InputVariables[2,86] AT %IB."KUKA3_KRC4_ProfiNet_5_0".Module001_8_digital_inputs_I_86;
	::InputVariables[2,87] AT %IB."KUKA3_KRC4_ProfiNet_5_0".Module001_8_digital_inputs_I_87;
	::InputVariables[2,88] AT %IB."KUKA3_KRC4_ProfiNet_5_0".Module001_8_digital_inputs_I_88;
	::InputVariables[2,89] AT %IB."KUKA3_KRC4_ProfiNet_5_0".Module001_8_digital_inputs_I_89;
	::InputVariables[2,90] AT %IB."KUKA3_KRC4_ProfiNet_5_0".Module001_8_digital_inputs_I_90;
	::InputVariables[2,91] AT %IB."KUKA3_KRC4_ProfiNet_5_0".Module001_8_digital_inputs_I_91;
	::InputVariables[2,92] AT %IB."KUKA3_KRC4_ProfiNet_5_0".Module001_8_digital_inputs_I_92;
	::InputVariables[2,93] AT %IB."KUKA3_KRC4_ProfiNet_5_0".Module001_8_digital_inputs_I_93;
	::InputVariables[2,94] AT %IB."KUKA3_KRC4_ProfiNet_5_0".Module001_8_digital_inputs_I_94;
	::InputVariables[2,95] AT %IB."KUKA3_KRC4_ProfiNet_5_0".Module001_8_digital_inputs_I_95;
	::InputVariables[2,96] AT %IB."KUKA3_KRC4_ProfiNet_5_0".Module001_8_digital_inputs_I_96;
	::InputVariables[2,97] AT %IB."KUKA3_KRC4_ProfiNet_5_0".Module001_8_digital_inputs_I_97;
	::InputVariables[2,98] AT %IB."KUKA3_KRC4_ProfiNet_5_0".Module001_8_digital_inputs_I_98;
	::InputVariables[2,99] AT %IB."KUKA3_KRC4_ProfiNet_5_0".Module001_8_digital_inputs_I_99;
	::InputVariables[2,100] AT %IB."KUKA3_KRC4_ProfiNet_5_0".Module001_8_digital_inputs_I_100;
	::InputVariables[2,101] AT %IB."KUKA3_KRC4_ProfiNet_5_0".Module001_8_digital_inputs_I_101;
	::InputVariables[2,102] AT %IB."KUKA3_KRC4_ProfiNet_5_0".Module001_8_digital_inputs_I_102;
	::InputVariables[2,103] AT %IB."KUKA3_KRC4_ProfiNet_5_0".Module001_8_digital_inputs_I_103;
	::InputVariables[2,104] AT %IB."KUKA3_KRC4_ProfiNet_5_0".Module001_8_digital_inputs_I_104;
	::InputVariables[2,105] AT %IB."KUKA3_KRC4_ProfiNet_5_0".Module001_8_digital_inputs_I_105;
	::InputVariables[2,106] AT %IB."KUKA3_KRC4_ProfiNet_5_0".Module001_8_digital_inputs_I_106;
	::InputVariables[2,107] AT %IB."KUKA3_KRC4_ProfiNet_5_0".Module001_8_digital_inputs_I_107;
	::InputVariables[2,108] AT %IB."KUKA3_KRC4_ProfiNet_5_0".Module001_8_digital_inputs_I_108;
	::InputVariables[2,109] AT %IB."KUKA3_KRC4_ProfiNet_5_0".Module001_8_digital_inputs_I_109;
	::InputVariables[2,110] AT %IB."KUKA3_KRC4_ProfiNet_5_0".Module001_8_digital_inputs_I_110;
	::InputVariables[2,111] AT %IB."KUKA3_KRC4_ProfiNet_5_0".Module001_8_digital_inputs_I_111;
	::InputVariables[2,112] AT %IB."KUKA3_KRC4_ProfiNet_5_0".Module001_8_digital_inputs_I_112;
	::InputVariables[2,113] AT %IB."KUKA3_KRC4_ProfiNet_5_0".Module001_8_digital_inputs_I_113;
	::InputVariables[2,114] AT %IB."KUKA3_KRC4_ProfiNet_5_0".Module001_8_digital_inputs_I_114;
	::InputVariables[2,115] AT %IB."KUKA3_KRC4_ProfiNet_5_0".Module001_8_digital_inputs_I_115;
	::InputVariables[2,116] AT %IB."KUKA3_KRC4_ProfiNet_5_0".Module001_8_digital_inputs_I_116;
	::InputVariables[2,117] AT %IB."KUKA3_KRC4_ProfiNet_5_0".Module001_8_digital_inputs_I_117;
	::InputVariables[2,118] AT %IB."KUKA3_KRC4_ProfiNet_5_0".Module001_8_digital_inputs_I_118;
	::InputVariables[2,119] AT %IB."KUKA3_KRC4_ProfiNet_5_0".Module001_8_digital_inputs_I_119;
	::InputVariables[2,120] AT %IB."KUKA3_KRC4_ProfiNet_5_0".Module001_8_digital_inputs_I_120;
	::InputVariables[2,121] AT %IB."KUKA3_KRC4_ProfiNet_5_0".Module001_8_digital_inputs_I_121;
	::InputVariables[2,122] AT %IB."KUKA3_KRC4_ProfiNet_5_0".Module001_8_digital_inputs_I_122;
	::InputVariables[2,123] AT %IB."KUKA3_KRC4_ProfiNet_5_0".Module001_8_digital_inputs_I_123;
	::InputVariables[2,124] AT %IB."KUKA3_KRC4_ProfiNet_5_0".Module001_8_digital_inputs_I_124;
	::InputVariables[2,125] AT %IB."KUKA3_KRC4_ProfiNet_5_0".Module001_8_digital_inputs_I_125;
	::InputVariables[2,126] AT %IB."KUKA3_KRC4_ProfiNet_5_0".Module001_8_digital_inputs_I_126;
	::InputVariables[2,127] AT %IB."KUKA3_KRC4_ProfiNet_5_0".Module001_8_digital_inputs_I_127;
	::InputVariables[2,128] AT %IB."KUKA3_KRC4_ProfiNet_5_0".Module001_8_digital_inputs_I_128;
	::InputVariables[2,129] AT %IB."KUKA3_KRC4_ProfiNet_5_0".Module001_8_digital_inputs_I_129;
	::InputVariables[2,130] AT %IB."KUKA3_KRC4_ProfiNet_5_0".Module001_8_digital_inputs_I_130;
	::InputVariables[2,131] AT %IB."KUKA3_KRC4_ProfiNet_5_0".Module001_8_digital_inputs_I_131;
	::InputVariables[2,132] AT %IB."KUKA3_KRC4_ProfiNet_5_0".Module001_8_digital_inputs_I_132;
	::InputVariables[2,133] AT %IB."KUKA3_KRC4_ProfiNet_5_0".Module001_8_digital_inputs_I_133;
	::InputVariables[2,134] AT %IB."KUKA3_KRC4_ProfiNet_5_0".Module001_8_digital_inputs_I_134;
	::InputVariables[2,135] AT %IB."KUKA3_KRC4_ProfiNet_5_0".Module001_8_digital_inputs_I_135;
	::InputVariables[2,136] AT %IB."KUKA3_KRC4_ProfiNet_5_0".Module001_8_digital_inputs_I_136;
	::InputVariables[2,137] AT %IB."KUKA3_KRC4_ProfiNet_5_0".Module001_8_digital_inputs_I_137;
	::InputVariables[2,138] AT %IB."KUKA3_KRC4_ProfiNet_5_0".Module001_8_digital_inputs_I_138;
	::InputVariables[2,139] AT %IB."KUKA3_KRC4_ProfiNet_5_0".Module001_8_digital_inputs_I_139;
	::InputVariables[2,140] AT %IB."KUKA3_KRC4_ProfiNet_5_0".Module001_8_digital_inputs_I_140;
	::InputVariables[2,141] AT %IB."KUKA3_KRC4_ProfiNet_5_0".Module001_8_digital_inputs_I_141;
	::InputVariables[2,142] AT %IB."KUKA3_KRC4_ProfiNet_5_0".Module001_8_digital_inputs_I_142;
	::InputVariables[2,143] AT %IB."KUKA3_KRC4_ProfiNet_5_0".Module001_8_digital_inputs_I_143;
	::InputVariables[2,144] AT %IB."KUKA3_KRC4_ProfiNet_5_0".Module001_8_digital_inputs_I_144;
	::InputVariables[2,145] AT %IB."KUKA3_KRC4_ProfiNet_5_0".Module001_8_digital_inputs_I_145;
	::InputVariables[2,146] AT %IB."KUKA3_KRC4_ProfiNet_5_0".Module001_8_digital_inputs_I_146;
	::InputVariables[2,147] AT %IB."KUKA3_KRC4_ProfiNet_5_0".Module001_8_digital_inputs_I_147;
	::InputVariables[2,148] AT %IB."KUKA3_KRC4_ProfiNet_5_0".Module001_8_digital_inputs_I_148;
	::InputVariables[2,149] AT %IB."KUKA3_KRC4_ProfiNet_5_0".Module001_8_digital_inputs_I_149;
	::InputVariables[2,150] AT %IB."KUKA3_KRC4_ProfiNet_5_0".Module001_8_digital_inputs_I_150;
	::InputVariables[2,151] AT %IB."KUKA3_KRC4_ProfiNet_5_0".Module001_8_digital_inputs_I_151;
	::InputVariables[2,152] AT %IB."KUKA3_KRC4_ProfiNet_5_0".Module001_8_digital_inputs_I_152;
	::InputVariables[2,153] AT %IB."KUKA3_KRC4_ProfiNet_5_0".Module001_8_digital_inputs_I_153;
	::InputVariables[2,154] AT %IB."KUKA3_KRC4_ProfiNet_5_0".Module001_8_digital_inputs_I_154;
	::InputVariables[2,155] AT %IB."KUKA3_KRC4_ProfiNet_5_0".Module001_8_digital_inputs_I_155;
	::InputVariables[2,156] AT %IB."KUKA3_KRC4_ProfiNet_5_0".Module001_8_digital_inputs_I_156;
	::InputVariables[2,157] AT %IB."KUKA3_KRC4_ProfiNet_5_0".Module001_8_digital_inputs_I_157;
	::InputVariables[2,158] AT %IB."KUKA3_KRC4_ProfiNet_5_0".Module001_8_digital_inputs_I_158;
	::InputVariables[2,159] AT %IB."KUKA3_KRC4_ProfiNet_5_0".Module001_8_digital_inputs_I_159;
	::InputVariables[2,160] AT %IB."KUKA3_KRC4_ProfiNet_5_0".Module001_8_digital_inputs_I_160;
	::InputVariables[2,161] AT %IB."KUKA3_KRC4_ProfiNet_5_0".Module001_8_digital_inputs_I_161;
	::InputVariables[2,162] AT %IB."KUKA3_KRC4_ProfiNet_5_0".Module001_8_digital_inputs_I_162;
	::InputVariables[2,163] AT %IB."KUKA3_KRC4_ProfiNet_5_0".Module001_8_digital_inputs_I_163;
	::InputVariables[2,164] AT %IB."KUKA3_KRC4_ProfiNet_5_0".Module001_8_digital_inputs_I_164;
	::InputVariables[2,165] AT %IB."KUKA3_KRC4_ProfiNet_5_0".Module001_8_digital_inputs_I_165;
	::InputVariables[2,166] AT %IB."KUKA3_KRC4_ProfiNet_5_0".Module001_8_digital_inputs_I_166;
	::InputVariables[2,167] AT %IB."KUKA3_KRC4_ProfiNet_5_0".Module001_8_digital_inputs_I_167;
	::InputVariables[2,168] AT %IB."KUKA3_KRC4_ProfiNet_5_0".Module001_8_digital_inputs_I_168;
	::InputVariables[2,169] AT %IB."KUKA3_KRC4_ProfiNet_5_0".Module001_8_digital_inputs_I_169;
	::InputVariables[2,170] AT %IB."KUKA3_KRC4_ProfiNet_5_0".Module001_8_digital_inputs_I_170;
	::InputVariables[2,171] AT %IB."KUKA3_KRC4_ProfiNet_5_0".Module001_8_digital_inputs_I_171;
	::InputVariables[2,172] AT %IB."KUKA3_KRC4_ProfiNet_5_0".Module001_8_digital_inputs_I_172;
	::InputVariables[2,173] AT %IB."KUKA3_KRC4_ProfiNet_5_0".Module001_8_digital_inputs_I_173;
	::InputVariables[2,174] AT %IB."KUKA3_KRC4_ProfiNet_5_0".Module001_8_digital_inputs_I_174;
	::InputVariables[2,175] AT %IB."KUKA3_KRC4_ProfiNet_5_0".Module001_8_digital_inputs_I_175;
	::InputVariables[2,176] AT %IB."KUKA3_KRC4_ProfiNet_5_0".Module001_8_digital_inputs_I_176;
	::InputVariables[2,177] AT %IB."KUKA3_KRC4_ProfiNet_5_0".Module001_8_digital_inputs_I_177;
	::InputVariables[2,178] AT %IB."KUKA3_KRC4_ProfiNet_5_0".Module001_8_digital_inputs_I_178;
	::InputVariables[2,179] AT %IB."KUKA3_KRC4_ProfiNet_5_0".Module001_8_digital_inputs_I_179;
	::InputVariables[2,180] AT %IB."KUKA3_KRC4_ProfiNet_5_0".Module001_8_digital_inputs_I_180;
	::InputVariables[2,181] AT %IB."KUKA3_KRC4_ProfiNet_5_0".Module001_8_digital_inputs_I_181;
	::InputVariables[2,182] AT %IB."KUKA3_KRC4_ProfiNet_5_0".Module001_8_digital_inputs_I_182;
	::InputVariables[2,183] AT %IB."KUKA3_KRC4_ProfiNet_5_0".Module001_8_digital_inputs_I_183;
	::InputVariables[2,184] AT %IB."KUKA3_KRC4_ProfiNet_5_0".Module001_8_digital_inputs_I_184;
	::InputVariables[2,185] AT %IB."KUKA3_KRC4_ProfiNet_5_0".Module001_8_digital_inputs_I_185;
	::InputVariables[2,186] AT %IB."KUKA3_KRC4_ProfiNet_5_0".Module001_8_digital_inputs_I_186;
	::InputVariables[2,187] AT %IB."KUKA3_KRC4_ProfiNet_5_0".Module001_8_digital_inputs_I_187;
	::InputVariables[2,188] AT %IB."KUKA3_KRC4_ProfiNet_5_0".Module001_8_digital_inputs_I_188;
	::InputVariables[2,189] AT %IB."KUKA3_KRC4_ProfiNet_5_0".Module001_8_digital_inputs_I_189;
	::InputVariables[2,190] AT %IB."KUKA3_KRC4_ProfiNet_5_0".Module001_8_digital_inputs_I_190;
	::InputVariables[2,191] AT %IB."KUKA3_KRC4_ProfiNet_5_0".Module001_8_digital_inputs_I_191;
	::InputVariables[2,192] AT %IB."KUKA3_KRC4_ProfiNet_5_0".Module001_8_digital_inputs_I_192;
	::InputVariables[2,193] AT %IB."KUKA3_KRC4_ProfiNet_5_0".Module001_8_digital_inputs_I_193;
	::InputVariables[2,194] AT %IB."KUKA3_KRC4_ProfiNet_5_0".Module001_8_digital_inputs_I_194;
	::InputVariables[2,195] AT %IB."KUKA3_KRC4_ProfiNet_5_0".Module001_8_digital_inputs_I_195;
	::InputVariables[2,196] AT %IB."KUKA3_KRC4_ProfiNet_5_0".Module001_8_digital_inputs_I_196;
	::InputVariables[2,197] AT %IB."KUKA3_KRC4_ProfiNet_5_0".Module001_8_digital_inputs_I_197;
	::InputVariables[2,198] AT %IB."KUKA3_KRC4_ProfiNet_5_0".Module001_8_digital_inputs_I_198;
	::InputVariables[2,199] AT %IB."KUKA3_KRC4_ProfiNet_5_0".Module001_8_digital_inputs_I_199;
	::InputVariables[2,200] AT %IB."KUKA3_KRC4_ProfiNet_5_0".Module001_8_digital_inputs_I_200;
	::InputVariables[2,201] AT %IB."KUKA3_KRC4_ProfiNet_5_0".Module001_8_digital_inputs_I_201;
	::InputVariables[2,202] AT %IB."KUKA3_KRC4_ProfiNet_5_0".Module001_8_digital_inputs_I_202;
	::InputVariables[2,203] AT %IB."KUKA3_KRC4_ProfiNet_5_0".Module001_8_digital_inputs_I_203;
	::InputVariables[2,204] AT %IB."KUKA3_KRC4_ProfiNet_5_0".Module001_8_digital_inputs_I_204;
	::InputVariables[2,205] AT %IB."KUKA3_KRC4_ProfiNet_5_0".Module001_8_digital_inputs_I_205;
	::InputVariables[2,206] AT %IB."KUKA3_KRC4_ProfiNet_5_0".Module001_8_digital_inputs_I_206;
	::InputVariables[2,207] AT %IB."KUKA3_KRC4_ProfiNet_5_0".Module001_8_digital_inputs_I_207;
	::InputVariables[2,208] AT %IB."KUKA3_KRC4_ProfiNet_5_0".Module001_8_digital_inputs_I_208;
	::InputVariables[2,209] AT %IB."KUKA3_KRC4_ProfiNet_5_0".Module001_8_digital_inputs_I_209;
	::InputVariables[2,210] AT %IB."KUKA3_KRC4_ProfiNet_5_0".Module001_8_digital_inputs_I_210;
	::InputVariables[2,211] AT %IB."KUKA3_KRC4_ProfiNet_5_0".Module001_8_digital_inputs_I_211;
	::InputVariables[2,212] AT %IB."KUKA3_KRC4_ProfiNet_5_0".Module001_8_digital_inputs_I_212;
	::InputVariables[2,213] AT %IB."KUKA3_KRC4_ProfiNet_5_0".Module001_8_digital_inputs_I_213;
	::InputVariables[2,214] AT %IB."KUKA3_KRC4_ProfiNet_5_0".Module001_8_digital_inputs_I_214;
	::InputVariables[2,215] AT %IB."KUKA3_KRC4_ProfiNet_5_0".Module001_8_digital_inputs_I_215;
	::InputVariables[2,216] AT %IB."KUKA3_KRC4_ProfiNet_5_0".Module001_8_digital_inputs_I_216;
	::InputVariables[2,217] AT %IB."KUKA3_KRC4_ProfiNet_5_0".Module001_8_digital_inputs_I_217;
	::InputVariables[2,218] AT %IB."KUKA3_KRC4_ProfiNet_5_0".Module001_8_digital_inputs_I_218;
	::InputVariables[2,219] AT %IB."KUKA3_KRC4_ProfiNet_5_0".Module001_8_digital_inputs_I_219;
	::InputVariables[2,220] AT %IB."KUKA3_KRC4_ProfiNet_5_0".Module001_8_digital_inputs_I_220;
	::InputVariables[2,221] AT %IB."KUKA3_KRC4_ProfiNet_5_0".Module001_8_digital_inputs_I_221;
	::InputVariables[2,222] AT %IB."KUKA3_KRC4_ProfiNet_5_0".Module001_8_digital_inputs_I_222;
	::InputVariables[2,223] AT %IB."KUKA3_KRC4_ProfiNet_5_0".Module001_8_digital_inputs_I_223;
	::InputVariables[2,224] AT %IB."KUKA3_KRC4_ProfiNet_5_0".Module001_8_digital_inputs_I_224;
	::InputVariables[2,225] AT %IB."KUKA3_KRC4_ProfiNet_5_0".Module001_8_digital_inputs_I_225;
	::InputVariables[2,226] AT %IB."KUKA3_KRC4_ProfiNet_5_0".Module001_8_digital_inputs_I_226;
	::InputVariables[2,227] AT %IB."KUKA3_KRC4_ProfiNet_5_0".Module001_8_digital_inputs_I_227;
	::InputVariables[2,228] AT %IB."KUKA3_KRC4_ProfiNet_5_0".Module001_8_digital_inputs_I_228;
	::InputVariables[2,229] AT %IB."KUKA3_KRC4_ProfiNet_5_0".Module001_8_digital_inputs_I_229;
	::InputVariables[2,230] AT %IB."KUKA3_KRC4_ProfiNet_5_0".Module001_8_digital_inputs_I_230;
	::InputVariables[2,231] AT %IB."KUKA3_KRC4_ProfiNet_5_0".Module001_8_digital_inputs_I_231;
	::InputVariables[2,232] AT %IB."KUKA3_KRC4_ProfiNet_5_0".Module001_8_digital_inputs_I_232;
	::InputVariables[2,233] AT %IB."KUKA3_KRC4_ProfiNet_5_0".Module001_8_digital_inputs_I_233;
	::InputVariables[2,234] AT %IB."KUKA3_KRC4_ProfiNet_5_0".Module001_8_digital_inputs_I_234;
	::InputVariables[2,235] AT %IB."KUKA3_KRC4_ProfiNet_5_0".Module001_8_digital_inputs_I_235;
	::InputVariables[2,236] AT %IB."KUKA3_KRC4_ProfiNet_5_0".Module001_8_digital_inputs_I_236;
	::InputVariables[2,237] AT %IB."KUKA3_KRC4_ProfiNet_5_0".Module001_8_digital_inputs_I_237;
	::InputVariables[2,238] AT %IB."KUKA3_KRC4_ProfiNet_5_0".Module001_8_digital_inputs_I_238;
	::InputVariables[2,239] AT %IB."KUKA3_KRC4_ProfiNet_5_0".Module001_8_digital_inputs_I_239;
	::InputVariables[2,240] AT %IB."KUKA3_KRC4_ProfiNet_5_0".Module001_8_digital_inputs_I_240;
	::InputVariables[2,241] AT %IB."KUKA3_KRC4_ProfiNet_5_0".Module001_8_digital_inputs_I_241;
	::InputVariables[2,242] AT %IB."KUKA3_KRC4_ProfiNet_5_0".Module001_8_digital_inputs_I_242;
	::InputVariables[2,243] AT %IB."KUKA3_KRC4_ProfiNet_5_0".Module001_8_digital_inputs_I_243;
	::InputVariables[2,244] AT %IB."KUKA3_KRC4_ProfiNet_5_0".Module001_8_digital_inputs_I_244;
	::InputVariables[2,245] AT %IB."KUKA3_KRC4_ProfiNet_5_0".Module001_8_digital_inputs_I_245;
	::InputVariables[2,246] AT %IB."KUKA3_KRC4_ProfiNet_5_0".Module001_8_digital_inputs_I_246;
	::InputVariables[2,247] AT %IB."KUKA3_KRC4_ProfiNet_5_0".Module001_8_digital_inputs_I_247;
	::InputVariables[2,248] AT %IB."KUKA3_KRC4_ProfiNet_5_0".Module001_8_digital_inputs_I_248;
	::InputVariables[2,249] AT %IB."KUKA3_KRC4_ProfiNet_5_0".Module001_8_digital_inputs_I_249;
	::InputVariables[2,250] AT %IB."KUKA3_KRC4_ProfiNet_5_0".Module001_8_digital_inputs_I_250;
	::InputVariables[2,251] AT %IB."KUKA3_KRC4_ProfiNet_5_0".Module001_8_digital_inputs_I_251;
	::InputVariables[2,252] AT %IB."KUKA3_KRC4_ProfiNet_5_0".Module001_8_digital_inputs_I_252;
	::InputVariables[2,253] AT %IB."KUKA3_KRC4_ProfiNet_5_0".Module001_8_digital_inputs_I_253;

	::OutputVariables[2,0]	AT %QB."KUKA3_KRC4_ProfiNet_5_0".Module001_8_digital_outputs_O_00;
	::OutputVariables[2,1]	AT %QB."KUKA3_KRC4_ProfiNet_5_0".Module001_8_digital_outputs_O_01;
	::OutputVariables[2,2]	AT %QB."KUKA3_KRC4_ProfiNet_5_0".Module001_8_digital_outputs_O_02;
	::OutputVariables[2,3]	AT %QB."KUKA3_KRC4_ProfiNet_5_0".Module001_8_digital_outputs_O_03;
	::OutputVariables[2,4]	AT %QB."KUKA3_KRC4_ProfiNet_5_0".Module001_8_digital_outputs_O_04;
	::OutputVariables[2,5]	AT %QB."KUKA3_KRC4_ProfiNet_5_0".Module001_8_digital_outputs_O_05;
	::OutputVariables[2,6]	AT %QB."KUKA3_KRC4_ProfiNet_5_0".Module001_8_digital_outputs_O_06;
	::OutputVariables[2,7]	AT %QB."KUKA3_KRC4_ProfiNet_5_0".Module001_8_digital_outputs_O_07;
	::OutputVariables[2,8]	AT %QB."KUKA3_KRC4_ProfiNet_5_0".Module001_8_digital_outputs_O_08;
	::OutputVariables[2,9]	AT %QB."KUKA3_KRC4_ProfiNet_5_0".Module001_8_digital_outputs_O_09;
	::OutputVariables[2,10]	AT %QB."KUKA3_KRC4_ProfiNet_5_0".Module001_8_digital_outputs_O_10;
	::OutputVariables[2,11]	AT %QB."KUKA3_KRC4_ProfiNet_5_0".Module001_8_digital_outputs_O_11;
	::OutputVariables[2,12]	AT %QB."KUKA3_KRC4_ProfiNet_5_0".Module001_8_digital_outputs_O_12;
	::OutputVariables[2,13]	AT %QB."KUKA3_KRC4_ProfiNet_5_0".Module001_8_digital_outputs_O_13;
	::OutputVariables[2,14]	AT %QB."KUKA3_KRC4_ProfiNet_5_0".Module001_8_digital_outputs_O_14;
	::OutputVariables[2,15]	AT %QB."KUKA3_KRC4_ProfiNet_5_0".Module001_8_digital_outputs_O_15;
	::OutputVariables[2,16]	AT %QB."KUKA3_KRC4_ProfiNet_5_0".Module001_8_digital_outputs_O_16;
	::OutputVariables[2,17]	AT %QB."KUKA3_KRC4_ProfiNet_5_0".Module001_8_digital_outputs_O_17;
	::OutputVariables[2,18]	AT %QB."KUKA3_KRC4_ProfiNet_5_0".Module001_8_digital_outputs_O_18;
	::OutputVariables[2,19]	AT %QB."KUKA3_KRC4_ProfiNet_5_0".Module001_8_digital_outputs_O_19;
	::OutputVariables[2,20]	AT %QB."KUKA3_KRC4_ProfiNet_5_0".Module001_8_digital_outputs_O_20;
	::OutputVariables[2,21]	AT %QB."KUKA3_KRC4_ProfiNet_5_0".Module001_8_digital_outputs_O_21;
	::OutputVariables[2,22]	AT %QB."KUKA3_KRC4_ProfiNet_5_0".Module001_8_digital_outputs_O_22;
	::OutputVariables[2,23]	AT %QB."KUKA3_KRC4_ProfiNet_5_0".Module001_8_digital_outputs_O_23;
	::OutputVariables[2,24]	AT %QB."KUKA3_KRC4_ProfiNet_5_0".Module001_8_digital_outputs_O_24;
	::OutputVariables[2,25]	AT %QB."KUKA3_KRC4_ProfiNet_5_0".Module001_8_digital_outputs_O_25;
	::OutputVariables[2,26]	AT %QB."KUKA3_KRC4_ProfiNet_5_0".Module001_8_digital_outputs_O_26;
	::OutputVariables[2,27]	AT %QB."KUKA3_KRC4_ProfiNet_5_0".Module001_8_digital_outputs_O_27;
	::OutputVariables[2,28]	AT %QB."KUKA3_KRC4_ProfiNet_5_0".Module001_8_digital_outputs_O_28;
	::OutputVariables[2,29]	AT %QB."KUKA3_KRC4_ProfiNet_5_0".Module001_8_digital_outputs_O_29;
	::OutputVariables[2,30]	AT %QB."KUKA3_KRC4_ProfiNet_5_0".Module001_8_digital_outputs_O_30;
	::OutputVariables[2,31]	AT %QB."KUKA3_KRC4_ProfiNet_5_0".Module001_8_digital_outputs_O_31;
	::OutputVariables[2,32]	AT %QB."KUKA3_KRC4_ProfiNet_5_0".Module001_8_digital_outputs_O_32;
	::OutputVariables[2,33]	AT %QB."KUKA3_KRC4_ProfiNet_5_0".Module001_8_digital_outputs_O_33;
	::OutputVariables[2,34]	AT %QB."KUKA3_KRC4_ProfiNet_5_0".Module001_8_digital_outputs_O_34;
	::OutputVariables[2,35]	AT %QB."KUKA3_KRC4_ProfiNet_5_0".Module001_8_digital_outputs_O_35;
	::OutputVariables[2,36]	AT %QB."KUKA3_KRC4_ProfiNet_5_0".Module001_8_digital_outputs_O_36;
	::OutputVariables[2,37]	AT %QB."KUKA3_KRC4_ProfiNet_5_0".Module001_8_digital_outputs_O_37;
	::OutputVariables[2,38]	AT %QB."KUKA3_KRC4_ProfiNet_5_0".Module001_8_digital_outputs_O_38;
	::OutputVariables[2,39]	AT %QB."KUKA3_KRC4_ProfiNet_5_0".Module001_8_digital_outputs_O_39;
	::OutputVariables[2,40]	AT %QB."KUKA3_KRC4_ProfiNet_5_0".Module001_8_digital_outputs_O_40;
	::OutputVariables[2,41]	AT %QB."KUKA3_KRC4_ProfiNet_5_0".Module001_8_digital_outputs_O_41;
	::OutputVariables[2,42]	AT %QB."KUKA3_KRC4_ProfiNet_5_0".Module001_8_digital_outputs_O_42;
	::OutputVariables[2,43]	AT %QB."KUKA3_KRC4_ProfiNet_5_0".Module001_8_digital_outputs_O_43;
	::OutputVariables[2,44]	AT %QB."KUKA3_KRC4_ProfiNet_5_0".Module001_8_digital_outputs_O_44;
	::OutputVariables[2,45]	AT %QB."KUKA3_KRC4_ProfiNet_5_0".Module001_8_digital_outputs_O_45;
	::OutputVariables[2,46]	AT %QB."KUKA3_KRC4_ProfiNet_5_0".Module001_8_digital_outputs_O_46;
	::OutputVariables[2,47]	AT %QB."KUKA3_KRC4_ProfiNet_5_0".Module001_8_digital_outputs_O_47;
	::OutputVariables[2,48]	AT %QB."KUKA3_KRC4_ProfiNet_5_0".Module001_8_digital_outputs_O_48;
	::OutputVariables[2,49]	AT %QB."KUKA3_KRC4_ProfiNet_5_0".Module001_8_digital_outputs_O_49;
	::OutputVariables[2,50]	AT %QB."KUKA3_KRC4_ProfiNet_5_0".Module001_8_digital_outputs_O_50;
	::OutputVariables[2,51]	AT %QB."KUKA3_KRC4_ProfiNet_5_0".Module001_8_digital_outputs_O_51;
	::OutputVariables[2,52]	AT %QB."KUKA3_KRC4_ProfiNet_5_0".Module001_8_digital_outputs_O_52;
	::OutputVariables[2,53]	AT %QB."KUKA3_KRC4_ProfiNet_5_0".Module001_8_digital_outputs_O_53;
	::OutputVariables[2,54]	AT %QB."KUKA3_KRC4_ProfiNet_5_0".Module001_8_digital_outputs_O_54;
	::OutputVariables[2,55]	AT %QB."KUKA3_KRC4_ProfiNet_5_0".Module001_8_digital_outputs_O_55;
	::OutputVariables[2,56]	AT %QB."KUKA3_KRC4_ProfiNet_5_0".Module001_8_digital_outputs_O_56;
	::OutputVariables[2,57]	AT %QB."KUKA3_KRC4_ProfiNet_5_0".Module001_8_digital_outputs_O_57;
	::OutputVariables[2,58]	AT %QB."KUKA3_KRC4_ProfiNet_5_0".Module001_8_digital_outputs_O_58;
	::OutputVariables[2,59]	AT %QB."KUKA3_KRC4_ProfiNet_5_0".Module001_8_digital_outputs_O_59;
	::OutputVariables[2,60]	AT %QB."KUKA3_KRC4_ProfiNet_5_0".Module001_8_digital_outputs_O_60;
	::OutputVariables[2,61]	AT %QB."KUKA3_KRC4_ProfiNet_5_0".Module001_8_digital_outputs_O_61;
	::OutputVariables[2,62]	AT %QB."KUKA3_KRC4_ProfiNet_5_0".Module001_8_digital_outputs_O_62;
	::OutputVariables[2,63]	AT %QB."KUKA3_KRC4_ProfiNet_5_0".Module001_8_digital_outputs_O_63;
	::OutputVariables[2,64]	AT %QB."KUKA3_KRC4_ProfiNet_5_0".Module001_8_digital_outputs_O_64;
	::OutputVariables[2,65]	AT %QB."KUKA3_KRC4_ProfiNet_5_0".Module001_8_digital_outputs_O_65;
	::OutputVariables[2,66]	AT %QB."KUKA3_KRC4_ProfiNet_5_0".Module001_8_digital_outputs_O_66;
	::OutputVariables[2,67]	AT %QB."KUKA3_KRC4_ProfiNet_5_0".Module001_8_digital_outputs_O_67;
	::OutputVariables[2,68]	AT %QB."KUKA3_KRC4_ProfiNet_5_0".Module001_8_digital_outputs_O_68;
	::OutputVariables[2,69]	AT %QB."KUKA3_KRC4_ProfiNet_5_0".Module001_8_digital_outputs_O_69;
	::OutputVariables[2,70]	AT %QB."KUKA3_KRC4_ProfiNet_5_0".Module001_8_digital_outputs_O_70;
	::OutputVariables[2,71]	AT %QB."KUKA3_KRC4_ProfiNet_5_0".Module001_8_digital_outputs_O_71;
	::OutputVariables[2,72]	AT %QB."KUKA3_KRC4_ProfiNet_5_0".Module001_8_digital_outputs_O_72;
	::OutputVariables[2,73]	AT %QB."KUKA3_KRC4_ProfiNet_5_0".Module001_8_digital_outputs_O_73;
	::OutputVariables[2,74]	AT %QB."KUKA3_KRC4_ProfiNet_5_0".Module001_8_digital_outputs_O_74;
	::OutputVariables[2,75]	AT %QB."KUKA3_KRC4_ProfiNet_5_0".Module001_8_digital_outputs_O_75;
	::OutputVariables[2,76]	AT %QB."KUKA3_KRC4_ProfiNet_5_0".Module001_8_digital_outputs_O_76;
	::OutputVariables[2,77]	AT %QB."KUKA3_KRC4_ProfiNet_5_0".Module001_8_digital_outputs_O_77;
	::OutputVariables[2,78]	AT %QB."KUKA3_KRC4_ProfiNet_5_0".Module001_8_digital_outputs_O_78;
	::OutputVariables[2,79]	AT %QB."KUKA3_KRC4_ProfiNet_5_0".Module001_8_digital_outputs_O_79;
	::OutputVariables[2,80]	AT %QB."KUKA3_KRC4_ProfiNet_5_0".Module001_8_digital_outputs_O_80;
	::OutputVariables[2,81]	AT %QB."KUKA3_KRC4_ProfiNet_5_0".Module001_8_digital_outputs_O_81;
	::OutputVariables[2,82]	AT %QB."KUKA3_KRC4_ProfiNet_5_0".Module001_8_digital_outputs_O_82;
	::OutputVariables[2,83]	AT %QB."KUKA3_KRC4_ProfiNet_5_0".Module001_8_digital_outputs_O_83;
	::OutputVariables[2,84]	AT %QB."KUKA3_KRC4_ProfiNet_5_0".Module001_8_digital_outputs_O_84;
	::OutputVariables[2,85]	AT %QB."KUKA3_KRC4_ProfiNet_5_0".Module001_8_digital_outputs_O_85;
	::OutputVariables[2,86]	AT %QB."KUKA3_KRC4_ProfiNet_5_0".Module001_8_digital_outputs_O_86;
	::OutputVariables[2,87]	AT %QB."KUKA3_KRC4_ProfiNet_5_0".Module001_8_digital_outputs_O_87;
	::OutputVariables[2,88]	AT %QB."KUKA3_KRC4_ProfiNet_5_0".Module001_8_digital_outputs_O_88;
	::OutputVariables[2,89]	AT %QB."KUKA3_KRC4_ProfiNet_5_0".Module001_8_digital_outputs_O_89;
	::OutputVariables[2,90]	AT %QB."KUKA3_KRC4_ProfiNet_5_0".Module001_8_digital_outputs_O_90;
	::OutputVariables[2,91]	AT %QB."KUKA3_KRC4_ProfiNet_5_0".Module001_8_digital_outputs_O_91;
	::OutputVariables[2,92]	AT %QB."KUKA3_KRC4_ProfiNet_5_0".Module001_8_digital_outputs_O_92;
	::OutputVariables[2,93]	AT %QB."KUKA3_KRC4_ProfiNet_5_0".Module001_8_digital_outputs_O_93;
	::OutputVariables[2,94]	AT %QB."KUKA3_KRC4_ProfiNet_5_0".Module001_8_digital_outputs_O_94;
	::OutputVariables[2,95]	AT %QB."KUKA3_KRC4_ProfiNet_5_0".Module001_8_digital_outputs_O_95;
	::OutputVariables[2,96]	AT %QB."KUKA3_KRC4_ProfiNet_5_0".Module001_8_digital_outputs_O_96;
	::OutputVariables[2,97]	AT %QB."KUKA3_KRC4_ProfiNet_5_0".Module001_8_digital_outputs_O_97;
	::OutputVariables[2,98]	AT %QB."KUKA3_KRC4_ProfiNet_5_0".Module001_8_digital_outputs_O_98;
	::OutputVariables[2,99]	AT %QB."KUKA3_KRC4_ProfiNet_5_0".Module001_8_digital_outputs_O_99;
	::OutputVariables[2,100]	AT %QB."KUKA3_KRC4_ProfiNet_5_0".Module001_8_digital_outputs_O_100;
	::OutputVariables[2,101]	AT %QB."KUKA3_KRC4_ProfiNet_5_0".Module001_8_digital_outputs_O_101;
	::OutputVariables[2,102]	AT %QB."KUKA3_KRC4_ProfiNet_5_0".Module001_8_digital_outputs_O_102;
	::OutputVariables[2,103]	AT %QB."KUKA3_KRC4_ProfiNet_5_0".Module001_8_digital_outputs_O_103;
	::OutputVariables[2,104]	AT %QB."KUKA3_KRC4_ProfiNet_5_0".Module001_8_digital_outputs_O_104;
	::OutputVariables[2,105]	AT %QB."KUKA3_KRC4_ProfiNet_5_0".Module001_8_digital_outputs_O_105;
	::OutputVariables[2,106]	AT %QB."KUKA3_KRC4_ProfiNet_5_0".Module001_8_digital_outputs_O_106;
	::OutputVariables[2,107]	AT %QB."KUKA3_KRC4_ProfiNet_5_0".Module001_8_digital_outputs_O_107;
	::OutputVariables[2,108]	AT %QB."KUKA3_KRC4_ProfiNet_5_0".Module001_8_digital_outputs_O_108;
	::OutputVariables[2,109]	AT %QB."KUKA3_KRC4_ProfiNet_5_0".Module001_8_digital_outputs_O_109;
	::OutputVariables[2,110]	AT %QB."KUKA3_KRC4_ProfiNet_5_0".Module001_8_digital_outputs_O_110;
	::OutputVariables[2,111]	AT %QB."KUKA3_KRC4_ProfiNet_5_0".Module001_8_digital_outputs_O_111;
	::OutputVariables[2,112]	AT %QB."KUKA3_KRC4_ProfiNet_5_0".Module001_8_digital_outputs_O_112;
	::OutputVariables[2,113]	AT %QB."KUKA3_KRC4_ProfiNet_5_0".Module001_8_digital_outputs_O_113;
	::OutputVariables[2,114]	AT %QB."KUKA3_KRC4_ProfiNet_5_0".Module001_8_digital_outputs_O_114;
	::OutputVariables[2,115]	AT %QB."KUKA3_KRC4_ProfiNet_5_0".Module001_8_digital_outputs_O_115;
	::OutputVariables[2,116]	AT %QB."KUKA3_KRC4_ProfiNet_5_0".Module001_8_digital_outputs_O_116;
	::OutputVariables[2,117]	AT %QB."KUKA3_KRC4_ProfiNet_5_0".Module001_8_digital_outputs_O_117;
	::OutputVariables[2,118]	AT %QB."KUKA3_KRC4_ProfiNet_5_0".Module001_8_digital_outputs_O_118;
	::OutputVariables[2,119]	AT %QB."KUKA3_KRC4_ProfiNet_5_0".Module001_8_digital_outputs_O_119;
	::OutputVariables[2,120]	AT %QB."KUKA3_KRC4_ProfiNet_5_0".Module001_8_digital_outputs_O_120;
	::OutputVariables[2,121]	AT %QB."KUKA3_KRC4_ProfiNet_5_0".Module001_8_digital_outputs_O_121;
	::OutputVariables[2,122]	AT %QB."KUKA3_KRC4_ProfiNet_5_0".Module001_8_digital_outputs_O_122;
	::OutputVariables[2,123]	AT %QB."KUKA3_KRC4_ProfiNet_5_0".Module001_8_digital_outputs_O_123;
	::OutputVariables[2,124]	AT %QB."KUKA3_KRC4_ProfiNet_5_0".Module001_8_digital_outputs_O_124;
	::OutputVariables[2,125]	AT %QB."KUKA3_KRC4_ProfiNet_5_0".Module001_8_digital_outputs_O_125;
	::OutputVariables[2,126]	AT %QB."KUKA3_KRC4_ProfiNet_5_0".Module001_8_digital_outputs_O_126;
	::OutputVariables[2,127]	AT %QB."KUKA3_KRC4_ProfiNet_5_0".Module001_8_digital_outputs_O_127;
	::OutputVariables[2,128]	AT %QB."KUKA3_KRC4_ProfiNet_5_0".Module001_8_digital_outputs_O_128;
	::OutputVariables[2,129]	AT %QB."KUKA3_KRC4_ProfiNet_5_0".Module001_8_digital_outputs_O_129;
	::OutputVariables[2,130]	AT %QB."KUKA3_KRC4_ProfiNet_5_0".Module001_8_digital_outputs_O_130;
	::OutputVariables[2,131]	AT %QB."KUKA3_KRC4_ProfiNet_5_0".Module001_8_digital_outputs_O_131;
	::OutputVariables[2,132]	AT %QB."KUKA3_KRC4_ProfiNet_5_0".Module001_8_digital_outputs_O_132;
	::OutputVariables[2,133]	AT %QB."KUKA3_KRC4_ProfiNet_5_0".Module001_8_digital_outputs_O_133;
	::OutputVariables[2,134]	AT %QB."KUKA3_KRC4_ProfiNet_5_0".Module001_8_digital_outputs_O_134;
	::OutputVariables[2,135]	AT %QB."KUKA3_KRC4_ProfiNet_5_0".Module001_8_digital_outputs_O_135;
	::OutputVariables[2,136]	AT %QB."KUKA3_KRC4_ProfiNet_5_0".Module001_8_digital_outputs_O_136;
	::OutputVariables[2,137]	AT %QB."KUKA3_KRC4_ProfiNet_5_0".Module001_8_digital_outputs_O_137;
	::OutputVariables[2,138]	AT %QB."KUKA3_KRC4_ProfiNet_5_0".Module001_8_digital_outputs_O_138;
	::OutputVariables[2,139]	AT %QB."KUKA3_KRC4_ProfiNet_5_0".Module001_8_digital_outputs_O_139;
	::OutputVariables[2,140]	AT %QB."KUKA3_KRC4_ProfiNet_5_0".Module001_8_digital_outputs_O_140;
	::OutputVariables[2,141]	AT %QB."KUKA3_KRC4_ProfiNet_5_0".Module001_8_digital_outputs_O_141;
	::OutputVariables[2,142]	AT %QB."KUKA3_KRC4_ProfiNet_5_0".Module001_8_digital_outputs_O_142;
	::OutputVariables[2,143]	AT %QB."KUKA3_KRC4_ProfiNet_5_0".Module001_8_digital_outputs_O_143;
	::OutputVariables[2,144]	AT %QB."KUKA3_KRC4_ProfiNet_5_0".Module001_8_digital_outputs_O_144;
	::OutputVariables[2,145]	AT %QB."KUKA3_KRC4_ProfiNet_5_0".Module001_8_digital_outputs_O_145;
	::OutputVariables[2,146]	AT %QB."KUKA3_KRC4_ProfiNet_5_0".Module001_8_digital_outputs_O_146;
	::OutputVariables[2,147]	AT %QB."KUKA3_KRC4_ProfiNet_5_0".Module001_8_digital_outputs_O_147;
	::OutputVariables[2,148]	AT %QB."KUKA3_KRC4_ProfiNet_5_0".Module001_8_digital_outputs_O_148;
	::OutputVariables[2,149]	AT %QB."KUKA3_KRC4_ProfiNet_5_0".Module001_8_digital_outputs_O_149;
	::OutputVariables[2,150]	AT %QB."KUKA3_KRC4_ProfiNet_5_0".Module001_8_digital_outputs_O_150;
	::OutputVariables[2,151]	AT %QB."KUKA3_KRC4_ProfiNet_5_0".Module001_8_digital_outputs_O_151;
	::OutputVariables[2,152]	AT %QB."KUKA3_KRC4_ProfiNet_5_0".Module001_8_digital_outputs_O_152;
	::OutputVariables[2,153]	AT %QB."KUKA3_KRC4_ProfiNet_5_0".Module001_8_digital_outputs_O_153;
	::OutputVariables[2,154]	AT %QB."KUKA3_KRC4_ProfiNet_5_0".Module001_8_digital_outputs_O_154;
	::OutputVariables[2,155]	AT %QB."KUKA3_KRC4_ProfiNet_5_0".Module001_8_digital_outputs_O_155;
	::OutputVariables[2,156]	AT %QB."KUKA3_KRC4_ProfiNet_5_0".Module001_8_digital_outputs_O_156;
	::OutputVariables[2,157]	AT %QB."KUKA3_KRC4_ProfiNet_5_0".Module001_8_digital_outputs_O_157;
	::OutputVariables[2,158]	AT %QB."KUKA3_KRC4_ProfiNet_5_0".Module001_8_digital_outputs_O_158;
	::OutputVariables[2,159]	AT %QB."KUKA3_KRC4_ProfiNet_5_0".Module001_8_digital_outputs_O_159;
	::OutputVariables[2,160]	AT %QB."KUKA3_KRC4_ProfiNet_5_0".Module001_8_digital_outputs_O_160;
	::OutputVariables[2,161]	AT %QB."KUKA3_KRC4_ProfiNet_5_0".Module001_8_digital_outputs_O_161;
	::OutputVariables[2,162]	AT %QB."KUKA3_KRC4_ProfiNet_5_0".Module001_8_digital_outputs_O_162;
	::OutputVariables[2,163]	AT %QB."KUKA3_KRC4_ProfiNet_5_0".Module001_8_digital_outputs_O_163;
	::OutputVariables[2,164]	AT %QB."KUKA3_KRC4_ProfiNet_5_0".Module001_8_digital_outputs_O_164;
	::OutputVariables[2,165]	AT %QB."KUKA3_KRC4_ProfiNet_5_0".Module001_8_digital_outputs_O_165;
	::OutputVariables[2,166]	AT %QB."KUKA3_KRC4_ProfiNet_5_0".Module001_8_digital_outputs_O_166;
	::OutputVariables[2,167]	AT %QB."KUKA3_KRC4_ProfiNet_5_0".Module001_8_digital_outputs_O_167;
	::OutputVariables[2,168]	AT %QB."KUKA3_KRC4_ProfiNet_5_0".Module001_8_digital_outputs_O_168;
	::OutputVariables[2,169]	AT %QB."KUKA3_KRC4_ProfiNet_5_0".Module001_8_digital_outputs_O_169;
	::OutputVariables[2,170]	AT %QB."KUKA3_KRC4_ProfiNet_5_0".Module001_8_digital_outputs_O_170;
	::OutputVariables[2,171]	AT %QB."KUKA3_KRC4_ProfiNet_5_0".Module001_8_digital_outputs_O_171;
	::OutputVariables[2,172]	AT %QB."KUKA3_KRC4_ProfiNet_5_0".Module001_8_digital_outputs_O_172;
	::OutputVariables[2,173]	AT %QB."KUKA3_KRC4_ProfiNet_5_0".Module001_8_digital_outputs_O_173;
	::OutputVariables[2,174]	AT %QB."KUKA3_KRC4_ProfiNet_5_0".Module001_8_digital_outputs_O_174;
	::OutputVariables[2,175]	AT %QB."KUKA3_KRC4_ProfiNet_5_0".Module001_8_digital_outputs_O_175;
	::OutputVariables[2,176]	AT %QB."KUKA3_KRC4_ProfiNet_5_0".Module001_8_digital_outputs_O_176;
	::OutputVariables[2,177]	AT %QB."KUKA3_KRC4_ProfiNet_5_0".Module001_8_digital_outputs_O_177;
	::OutputVariables[2,178]	AT %QB."KUKA3_KRC4_ProfiNet_5_0".Module001_8_digital_outputs_O_178;
	::OutputVariables[2,179]	AT %QB."KUKA3_KRC4_ProfiNet_5_0".Module001_8_digital_outputs_O_179;
	::OutputVariables[2,180]	AT %QB."KUKA3_KRC4_ProfiNet_5_0".Module001_8_digital_outputs_O_180;
	::OutputVariables[2,181]	AT %QB."KUKA3_KRC4_ProfiNet_5_0".Module001_8_digital_outputs_O_181;
	::OutputVariables[2,182]	AT %QB."KUKA3_KRC4_ProfiNet_5_0".Module001_8_digital_outputs_O_182;
	::OutputVariables[2,183]	AT %QB."KUKA3_KRC4_ProfiNet_5_0".Module001_8_digital_outputs_O_183;
	::OutputVariables[2,184]	AT %QB."KUKA3_KRC4_ProfiNet_5_0".Module001_8_digital_outputs_O_184;
	::OutputVariables[2,185]	AT %QB."KUKA3_KRC4_ProfiNet_5_0".Module001_8_digital_outputs_O_185;
	::OutputVariables[2,186]	AT %QB."KUKA3_KRC4_ProfiNet_5_0".Module001_8_digital_outputs_O_186;
	::OutputVariables[2,187]	AT %QB."KUKA3_KRC4_ProfiNet_5_0".Module001_8_digital_outputs_O_187;
	::OutputVariables[2,188]	AT %QB."KUKA3_KRC4_ProfiNet_5_0".Module001_8_digital_outputs_O_188;
	::OutputVariables[2,189]	AT %QB."KUKA3_KRC4_ProfiNet_5_0".Module001_8_digital_outputs_O_189;
	::OutputVariables[2,190]	AT %QB."KUKA3_KRC4_ProfiNet_5_0".Module001_8_digital_outputs_O_190;
	::OutputVariables[2,191]	AT %QB."KUKA3_KRC4_ProfiNet_5_0".Module001_8_digital_outputs_O_191;
	::OutputVariables[2,192]	AT %QB."KUKA3_KRC4_ProfiNet_5_0".Module001_8_digital_outputs_O_192;
	::OutputVariables[2,193]	AT %QB."KUKA3_KRC4_ProfiNet_5_0".Module001_8_digital_outputs_O_193;
	::OutputVariables[2,194]	AT %QB."KUKA3_KRC4_ProfiNet_5_0".Module001_8_digital_outputs_O_194;
	::OutputVariables[2,195]	AT %QB."KUKA3_KRC4_ProfiNet_5_0".Module001_8_digital_outputs_O_195;
	::OutputVariables[2,196]	AT %QB."KUKA3_KRC4_ProfiNet_5_0".Module001_8_digital_outputs_O_196;
	::OutputVariables[2,197]	AT %QB."KUKA3_KRC4_ProfiNet_5_0".Module001_8_digital_outputs_O_197;
	::OutputVariables[2,198]	AT %QB."KUKA3_KRC4_ProfiNet_5_0".Module001_8_digital_outputs_O_198;
	::OutputVariables[2,199]	AT %QB."KUKA3_KRC4_ProfiNet_5_0".Module001_8_digital_outputs_O_199;
	::OutputVariables[2,200]	AT %QB."KUKA3_KRC4_ProfiNet_5_0".Module001_8_digital_outputs_O_200;
	::OutputVariables[2,201]	AT %QB."KUKA3_KRC4_ProfiNet_5_0".Module001_8_digital_outputs_O_201;
	::OutputVariables[2,202]	AT %QB."KUKA3_KRC4_ProfiNet_5_0".Module001_8_digital_outputs_O_202;
	::OutputVariables[2,203]	AT %QB."KUKA3_KRC4_ProfiNet_5_0".Module001_8_digital_outputs_O_203;
	::OutputVariables[2,204]	AT %QB."KUKA3_KRC4_ProfiNet_5_0".Module001_8_digital_outputs_O_204;
	::OutputVariables[2,205]	AT %QB."KUKA3_KRC4_ProfiNet_5_0".Module001_8_digital_outputs_O_205;
	::OutputVariables[2,206]	AT %QB."KUKA3_KRC4_ProfiNet_5_0".Module001_8_digital_outputs_O_206;
	::OutputVariables[2,207]	AT %QB."KUKA3_KRC4_ProfiNet_5_0".Module001_8_digital_outputs_O_207;
	::OutputVariables[2,208]	AT %QB."KUKA3_KRC4_ProfiNet_5_0".Module001_8_digital_outputs_O_208;
	::OutputVariables[2,209]	AT %QB."KUKA3_KRC4_ProfiNet_5_0".Module001_8_digital_outputs_O_209;
	::OutputVariables[2,210]	AT %QB."KUKA3_KRC4_ProfiNet_5_0".Module001_8_digital_outputs_O_210;
	::OutputVariables[2,211]	AT %QB."KUKA3_KRC4_ProfiNet_5_0".Module001_8_digital_outputs_O_211;
	::OutputVariables[2,212]	AT %QB."KUKA3_KRC4_ProfiNet_5_0".Module001_8_digital_outputs_O_212;
	::OutputVariables[2,213]	AT %QB."KUKA3_KRC4_ProfiNet_5_0".Module001_8_digital_outputs_O_213;
	::OutputVariables[2,214]	AT %QB."KUKA3_KRC4_ProfiNet_5_0".Module001_8_digital_outputs_O_214;
	::OutputVariables[2,215]	AT %QB."KUKA3_KRC4_ProfiNet_5_0".Module001_8_digital_outputs_O_215;
	::OutputVariables[2,216]	AT %QB."KUKA3_KRC4_ProfiNet_5_0".Module001_8_digital_outputs_O_216;
	::OutputVariables[2,217]	AT %QB."KUKA3_KRC4_ProfiNet_5_0".Module001_8_digital_outputs_O_217;
	::OutputVariables[2,218]	AT %QB."KUKA3_KRC4_ProfiNet_5_0".Module001_8_digital_outputs_O_218;
	::OutputVariables[2,219]	AT %QB."KUKA3_KRC4_ProfiNet_5_0".Module001_8_digital_outputs_O_219;
	::OutputVariables[2,220]	AT %QB."KUKA3_KRC4_ProfiNet_5_0".Module001_8_digital_outputs_O_220;
	::OutputVariables[2,221]	AT %QB."KUKA3_KRC4_ProfiNet_5_0".Module001_8_digital_outputs_O_221;
	::OutputVariables[2,222]	AT %QB."KUKA3_KRC4_ProfiNet_5_0".Module001_8_digital_outputs_O_222;
	::OutputVariables[2,223]	AT %QB."KUKA3_KRC4_ProfiNet_5_0".Module001_8_digital_outputs_O_223;
	::OutputVariables[2,224]	AT %QB."KUKA3_KRC4_ProfiNet_5_0".Module001_8_digital_outputs_O_224;
	::OutputVariables[2,225]	AT %QB."KUKA3_KRC4_ProfiNet_5_0".Module001_8_digital_outputs_O_225;
	::OutputVariables[2,226]	AT %QB."KUKA3_KRC4_ProfiNet_5_0".Module001_8_digital_outputs_O_226;
	::OutputVariables[2,227]	AT %QB."KUKA3_KRC4_ProfiNet_5_0".Module001_8_digital_outputs_O_227;
	::OutputVariables[2,228]	AT %QB."KUKA3_KRC4_ProfiNet_5_0".Module001_8_digital_outputs_O_228;
	::OutputVariables[2,229]	AT %QB."KUKA3_KRC4_ProfiNet_5_0".Module001_8_digital_outputs_O_229;
	::OutputVariables[2,230]	AT %QB."KUKA3_KRC4_ProfiNet_5_0".Module001_8_digital_outputs_O_230;
	::OutputVariables[2,231]	AT %QB."KUKA3_KRC4_ProfiNet_5_0".Module001_8_digital_outputs_O_231;
	::OutputVariables[2,232]	AT %QB."KUKA3_KRC4_ProfiNet_5_0".Module001_8_digital_outputs_O_232;
	::OutputVariables[2,233]	AT %QB."KUKA3_KRC4_ProfiNet_5_0".Module001_8_digital_outputs_O_233;
	::OutputVariables[2,234]	AT %QB."KUKA3_KRC4_ProfiNet_5_0".Module001_8_digital_outputs_O_234;
	::OutputVariables[2,235]	AT %QB."KUKA3_KRC4_ProfiNet_5_0".Module001_8_digital_outputs_O_235;
	::OutputVariables[2,236]	AT %QB."KUKA3_KRC4_ProfiNet_5_0".Module001_8_digital_outputs_O_236;
	::OutputVariables[2,237]	AT %QB."KUKA3_KRC4_ProfiNet_5_0".Module001_8_digital_outputs_O_237;
	::OutputVariables[2,238]	AT %QB."KUKA3_KRC4_ProfiNet_5_0".Module001_8_digital_outputs_O_238;
	::OutputVariables[2,239]	AT %QB."KUKA3_KRC4_ProfiNet_5_0".Module001_8_digital_outputs_O_239;
	::OutputVariables[2,240]	AT %QB."KUKA3_KRC4_ProfiNet_5_0".Module001_8_digital_outputs_O_240;
	::OutputVariables[2,241]	AT %QB."KUKA3_KRC4_ProfiNet_5_0".Module001_8_digital_outputs_O_241;
	::OutputVariables[2,242]	AT %QB."KUKA3_KRC4_ProfiNet_5_0".Module001_8_digital_outputs_O_242;
	::OutputVariables[2,243]	AT %QB."KUKA3_KRC4_ProfiNet_5_0".Module001_8_digital_outputs_O_243;
	::OutputVariables[2,244]	AT %QB."KUKA3_KRC4_ProfiNet_5_0".Module001_8_digital_outputs_O_244;
	::OutputVariables[2,245]	AT %QB."KUKA3_KRC4_ProfiNet_5_0".Module001_8_digital_outputs_O_245;
	::OutputVariables[2,246]	AT %QB."KUKA3_KRC4_ProfiNet_5_0".Module001_8_digital_outputs_O_246;
	::OutputVariables[2,247]	AT %QB."KUKA3_KRC4_ProfiNet_5_0".Module001_8_digital_outputs_O_247;
	::OutputVariables[2,248]	AT %QB."KUKA3_KRC4_ProfiNet_5_0".Module001_8_digital_outputs_O_248;
	::OutputVariables[2,249]	AT %QB."KUKA3_KRC4_ProfiNet_5_0".Module001_8_digital_outputs_O_249;
	::OutputVariables[2,250]	AT %QB."KUKA3_KRC4_ProfiNet_5_0".Module001_8_digital_outputs_O_250;
	::OutputVariables[2,251]	AT %QB."KUKA3_KRC4_ProfiNet_5_0".Module001_8_digital_outputs_O_251;
	::OutputVariables[2,252]	AT %QB."KUKA3_KRC4_ProfiNet_5_0".Module001_8_digital_outputs_O_252;
	::OutputVariables[2,253]	AT %QB."KUKA3_KRC4_ProfiNet_5_0".Module001_8_digital_outputs_O_253;

	(*________________________________________*)
	(*_____________KUKA4 Mappings_____________*)
	(*________________________________________*)

	::InputVariables[3,0] AT %IB."KUKA4_KRC4_ProfiNet_5_0".Module001_8_digital_inputs_I_00;
	::InputVariables[3,1] AT %IB."KUKA4_KRC4_ProfiNet_5_0".Module001_8_digital_inputs_I_01;
	::InputVariables[3,2] AT %IB."KUKA4_KRC4_ProfiNet_5_0".Module001_8_digital_inputs_I_02;
	::InputVariables[3,3] AT %IB."KUKA4_KRC4_ProfiNet_5_0".Module001_8_digital_inputs_I_03;
	::InputVariables[3,4] AT %IB."KUKA4_KRC4_ProfiNet_5_0".Module001_8_digital_inputs_I_04;
	::InputVariables[3,5] AT %IB."KUKA4_KRC4_ProfiNet_5_0".Module001_8_digital_inputs_I_05;
	::InputVariables[3,6] AT %IB."KUKA4_KRC4_ProfiNet_5_0".Module001_8_digital_inputs_I_06;
	::InputVariables[3,7] AT %IB."KUKA4_KRC4_ProfiNet_5_0".Module001_8_digital_inputs_I_07;
	::InputVariables[3,8] AT %IB."KUKA4_KRC4_ProfiNet_5_0".Module001_8_digital_inputs_I_08;
	::InputVariables[3,9] AT %IB."KUKA4_KRC4_ProfiNet_5_0".Module001_8_digital_inputs_I_09;
	::InputVariables[3,10] AT %IB."KUKA4_KRC4_ProfiNet_5_0".Module001_8_digital_inputs_I_10;
	::InputVariables[3,11] AT %IB."KUKA4_KRC4_ProfiNet_5_0".Module001_8_digital_inputs_I_11;
	::InputVariables[3,12] AT %IB."KUKA4_KRC4_ProfiNet_5_0".Module001_8_digital_inputs_I_12;
	::InputVariables[3,13] AT %IB."KUKA4_KRC4_ProfiNet_5_0".Module001_8_digital_inputs_I_13;
	::InputVariables[3,14] AT %IB."KUKA4_KRC4_ProfiNet_5_0".Module001_8_digital_inputs_I_14;
	::InputVariables[3,15] AT %IB."KUKA4_KRC4_ProfiNet_5_0".Module001_8_digital_inputs_I_15;
	::InputVariables[3,16] AT %IB."KUKA4_KRC4_ProfiNet_5_0".Module001_8_digital_inputs_I_16;
	::InputVariables[3,17] AT %IB."KUKA4_KRC4_ProfiNet_5_0".Module001_8_digital_inputs_I_17;
	::InputVariables[3,18] AT %IB."KUKA4_KRC4_ProfiNet_5_0".Module001_8_digital_inputs_I_18;
	::InputVariables[3,19] AT %IB."KUKA4_KRC4_ProfiNet_5_0".Module001_8_digital_inputs_I_19;
	::InputVariables[3,20] AT %IB."KUKA4_KRC4_ProfiNet_5_0".Module001_8_digital_inputs_I_20;
	::InputVariables[3,21] AT %IB."KUKA4_KRC4_ProfiNet_5_0".Module001_8_digital_inputs_I_21;
	::InputVariables[3,22] AT %IB."KUKA4_KRC4_ProfiNet_5_0".Module001_8_digital_inputs_I_22;
	::InputVariables[3,23] AT %IB."KUKA4_KRC4_ProfiNet_5_0".Module001_8_digital_inputs_I_23;
	::InputVariables[3,24] AT %IB."KUKA4_KRC4_ProfiNet_5_0".Module001_8_digital_inputs_I_24;
	::InputVariables[3,25] AT %IB."KUKA4_KRC4_ProfiNet_5_0".Module001_8_digital_inputs_I_25;
	::InputVariables[3,26] AT %IB."KUKA4_KRC4_ProfiNet_5_0".Module001_8_digital_inputs_I_26;
	::InputVariables[3,27] AT %IB."KUKA4_KRC4_ProfiNet_5_0".Module001_8_digital_inputs_I_27;
	::InputVariables[3,28] AT %IB."KUKA4_KRC4_ProfiNet_5_0".Module001_8_digital_inputs_I_28;
	::InputVariables[3,29] AT %IB."KUKA4_KRC4_ProfiNet_5_0".Module001_8_digital_inputs_I_29;
	::InputVariables[3,30] AT %IB."KUKA4_KRC4_ProfiNet_5_0".Module001_8_digital_inputs_I_30;
	::InputVariables[3,31] AT %IB."KUKA4_KRC4_ProfiNet_5_0".Module001_8_digital_inputs_I_31;
	::InputVariables[3,32] AT %IB."KUKA4_KRC4_ProfiNet_5_0".Module001_8_digital_inputs_I_32;
	::InputVariables[3,33] AT %IB."KUKA4_KRC4_ProfiNet_5_0".Module001_8_digital_inputs_I_33;
	::InputVariables[3,34] AT %IB."KUKA4_KRC4_ProfiNet_5_0".Module001_8_digital_inputs_I_34;
	::InputVariables[3,35] AT %IB."KUKA4_KRC4_ProfiNet_5_0".Module001_8_digital_inputs_I_35;
	::InputVariables[3,36] AT %IB."KUKA4_KRC4_ProfiNet_5_0".Module001_8_digital_inputs_I_36;
	::InputVariables[3,37] AT %IB."KUKA4_KRC4_ProfiNet_5_0".Module001_8_digital_inputs_I_37;
	::InputVariables[3,38] AT %IB."KUKA4_KRC4_ProfiNet_5_0".Module001_8_digital_inputs_I_38;
	::InputVariables[3,39] AT %IB."KUKA4_KRC4_ProfiNet_5_0".Module001_8_digital_inputs_I_39;
	::InputVariables[3,40] AT %IB."KUKA4_KRC4_ProfiNet_5_0".Module001_8_digital_inputs_I_40;
	::InputVariables[3,41] AT %IB."KUKA4_KRC4_ProfiNet_5_0".Module001_8_digital_inputs_I_41;
	::InputVariables[3,42] AT %IB."KUKA4_KRC4_ProfiNet_5_0".Module001_8_digital_inputs_I_42;
	::InputVariables[3,43] AT %IB."KUKA4_KRC4_ProfiNet_5_0".Module001_8_digital_inputs_I_43;
	::InputVariables[3,44] AT %IB."KUKA4_KRC4_ProfiNet_5_0".Module001_8_digital_inputs_I_44;
	::InputVariables[3,45] AT %IB."KUKA4_KRC4_ProfiNet_5_0".Module001_8_digital_inputs_I_45;
	::InputVariables[3,46] AT %IB."KUKA4_KRC4_ProfiNet_5_0".Module001_8_digital_inputs_I_46;
	::InputVariables[3,47] AT %IB."KUKA4_KRC4_ProfiNet_5_0".Module001_8_digital_inputs_I_47;
	::InputVariables[3,48] AT %IB."KUKA4_KRC4_ProfiNet_5_0".Module001_8_digital_inputs_I_48;
	::InputVariables[3,49] AT %IB."KUKA4_KRC4_ProfiNet_5_0".Module001_8_digital_inputs_I_49;
	::InputVariables[3,50] AT %IB."KUKA4_KRC4_ProfiNet_5_0".Module001_8_digital_inputs_I_50;
	::InputVariables[3,51] AT %IB."KUKA4_KRC4_ProfiNet_5_0".Module001_8_digital_inputs_I_51;
	::InputVariables[3,52] AT %IB."KUKA4_KRC4_ProfiNet_5_0".Module001_8_digital_inputs_I_52;
	::InputVariables[3,53] AT %IB."KUKA4_KRC4_ProfiNet_5_0".Module001_8_digital_inputs_I_53;
	::InputVariables[3,54] AT %IB."KUKA4_KRC4_ProfiNet_5_0".Module001_8_digital_inputs_I_54;
	::InputVariables[3,55] AT %IB."KUKA4_KRC4_ProfiNet_5_0".Module001_8_digital_inputs_I_55;
	::InputVariables[3,56] AT %IB."KUKA4_KRC4_ProfiNet_5_0".Module001_8_digital_inputs_I_56;
	::InputVariables[3,57] AT %IB."KUKA4_KRC4_ProfiNet_5_0".Module001_8_digital_inputs_I_57;
	::InputVariables[3,58] AT %IB."KUKA4_KRC4_ProfiNet_5_0".Module001_8_digital_inputs_I_58;
	::InputVariables[3,59] AT %IB."KUKA4_KRC4_ProfiNet_5_0".Module001_8_digital_inputs_I_59;
	::InputVariables[3,60] AT %IB."KUKA4_KRC4_ProfiNet_5_0".Module001_8_digital_inputs_I_60;
	::InputVariables[3,61] AT %IB."KUKA4_KRC4_ProfiNet_5_0".Module001_8_digital_inputs_I_61;
	::InputVariables[3,62] AT %IB."KUKA4_KRC4_ProfiNet_5_0".Module001_8_digital_inputs_I_62;
	::InputVariables[3,63] AT %IB."KUKA4_KRC4_ProfiNet_5_0".Module001_8_digital_inputs_I_63;
	::InputVariables[3,64] AT %IB."KUKA4_KRC4_ProfiNet_5_0".Module001_8_digital_inputs_I_64;
	::InputVariables[3,65] AT %IB."KUKA4_KRC4_ProfiNet_5_0".Module001_8_digital_inputs_I_65;
	::InputVariables[3,66] AT %IB."KUKA4_KRC4_ProfiNet_5_0".Module001_8_digital_inputs_I_66;
	::InputVariables[3,67] AT %IB."KUKA4_KRC4_ProfiNet_5_0".Module001_8_digital_inputs_I_67;
	::InputVariables[3,68] AT %IB."KUKA4_KRC4_ProfiNet_5_0".Module001_8_digital_inputs_I_68;
	::InputVariables[3,69] AT %IB."KUKA4_KRC4_ProfiNet_5_0".Module001_8_digital_inputs_I_69;
	::InputVariables[3,70] AT %IB."KUKA4_KRC4_ProfiNet_5_0".Module001_8_digital_inputs_I_70;
	::InputVariables[3,71] AT %IB."KUKA4_KRC4_ProfiNet_5_0".Module001_8_digital_inputs_I_71;
	::InputVariables[3,72] AT %IB."KUKA4_KRC4_ProfiNet_5_0".Module001_8_digital_inputs_I_72;
	::InputVariables[3,73] AT %IB."KUKA4_KRC4_ProfiNet_5_0".Module001_8_digital_inputs_I_73;
	::InputVariables[3,74] AT %IB."KUKA4_KRC4_ProfiNet_5_0".Module001_8_digital_inputs_I_74;
	::InputVariables[3,75] AT %IB."KUKA4_KRC4_ProfiNet_5_0".Module001_8_digital_inputs_I_75;
	::InputVariables[3,76] AT %IB."KUKA4_KRC4_ProfiNet_5_0".Module001_8_digital_inputs_I_76;
	::InputVariables[3,77] AT %IB."KUKA4_KRC4_ProfiNet_5_0".Module001_8_digital_inputs_I_77;
	::InputVariables[3,78] AT %IB."KUKA4_KRC4_ProfiNet_5_0".Module001_8_digital_inputs_I_78;
	::InputVariables[3,79] AT %IB."KUKA4_KRC4_ProfiNet_5_0".Module001_8_digital_inputs_I_79;
	::InputVariables[3,80] AT %IB."KUKA4_KRC4_ProfiNet_5_0".Module001_8_digital_inputs_I_80;
	::InputVariables[3,81] AT %IB."KUKA4_KRC4_ProfiNet_5_0".Module001_8_digital_inputs_I_81;
	::InputVariables[3,82] AT %IB."KUKA4_KRC4_ProfiNet_5_0".Module001_8_digital_inputs_I_82;
	::InputVariables[3,83] AT %IB."KUKA4_KRC4_ProfiNet_5_0".Module001_8_digital_inputs_I_83;
	::InputVariables[3,84] AT %IB."KUKA4_KRC4_ProfiNet_5_0".Module001_8_digital_inputs_I_84;
	::InputVariables[3,85] AT %IB."KUKA4_KRC4_ProfiNet_5_0".Module001_8_digital_inputs_I_85;
	::InputVariables[3,86] AT %IB."KUKA4_KRC4_ProfiNet_5_0".Module001_8_digital_inputs_I_86;
	::InputVariables[3,87] AT %IB."KUKA4_KRC4_ProfiNet_5_0".Module001_8_digital_inputs_I_87;
	::InputVariables[3,88] AT %IB."KUKA4_KRC4_ProfiNet_5_0".Module001_8_digital_inputs_I_88;
	::InputVariables[3,89] AT %IB."KUKA4_KRC4_ProfiNet_5_0".Module001_8_digital_inputs_I_89;
	::InputVariables[3,90] AT %IB."KUKA4_KRC4_ProfiNet_5_0".Module001_8_digital_inputs_I_90;
	::InputVariables[3,91] AT %IB."KUKA4_KRC4_ProfiNet_5_0".Module001_8_digital_inputs_I_91;
	::InputVariables[3,92] AT %IB."KUKA4_KRC4_ProfiNet_5_0".Module001_8_digital_inputs_I_92;
	::InputVariables[3,93] AT %IB."KUKA4_KRC4_ProfiNet_5_0".Module001_8_digital_inputs_I_93;
	::InputVariables[3,94] AT %IB."KUKA4_KRC4_ProfiNet_5_0".Module001_8_digital_inputs_I_94;
	::InputVariables[3,95] AT %IB."KUKA4_KRC4_ProfiNet_5_0".Module001_8_digital_inputs_I_95;
	::InputVariables[3,96] AT %IB."KUKA4_KRC4_ProfiNet_5_0".Module001_8_digital_inputs_I_96;
	::InputVariables[3,97] AT %IB."KUKA4_KRC4_ProfiNet_5_0".Module001_8_digital_inputs_I_97;
	::InputVariables[3,98] AT %IB."KUKA4_KRC4_ProfiNet_5_0".Module001_8_digital_inputs_I_98;
	::InputVariables[3,99] AT %IB."KUKA4_KRC4_ProfiNet_5_0".Module001_8_digital_inputs_I_99;
	::InputVariables[3,100] AT %IB."KUKA4_KRC4_ProfiNet_5_0".Module001_8_digital_inputs_I_100;
	::InputVariables[3,101] AT %IB."KUKA4_KRC4_ProfiNet_5_0".Module001_8_digital_inputs_I_101;
	::InputVariables[3,102] AT %IB."KUKA4_KRC4_ProfiNet_5_0".Module001_8_digital_inputs_I_102;
	::InputVariables[3,103] AT %IB."KUKA4_KRC4_ProfiNet_5_0".Module001_8_digital_inputs_I_103;
	::InputVariables[3,104] AT %IB."KUKA4_KRC4_ProfiNet_5_0".Module001_8_digital_inputs_I_104;
	::InputVariables[3,105] AT %IB."KUKA4_KRC4_ProfiNet_5_0".Module001_8_digital_inputs_I_105;
	::InputVariables[3,106] AT %IB."KUKA4_KRC4_ProfiNet_5_0".Module001_8_digital_inputs_I_106;
	::InputVariables[3,107] AT %IB."KUKA4_KRC4_ProfiNet_5_0".Module001_8_digital_inputs_I_107;
	::InputVariables[3,108] AT %IB."KUKA4_KRC4_ProfiNet_5_0".Module001_8_digital_inputs_I_108;
	::InputVariables[3,109] AT %IB."KUKA4_KRC4_ProfiNet_5_0".Module001_8_digital_inputs_I_109;
	::InputVariables[3,110] AT %IB."KUKA4_KRC4_ProfiNet_5_0".Module001_8_digital_inputs_I_110;
	::InputVariables[3,111] AT %IB."KUKA4_KRC4_ProfiNet_5_0".Module001_8_digital_inputs_I_111;
	::InputVariables[3,112] AT %IB."KUKA4_KRC4_ProfiNet_5_0".Module001_8_digital_inputs_I_112;
	::InputVariables[3,113] AT %IB."KUKA4_KRC4_ProfiNet_5_0".Module001_8_digital_inputs_I_113;
	::InputVariables[3,114] AT %IB."KUKA4_KRC4_ProfiNet_5_0".Module001_8_digital_inputs_I_114;
	::InputVariables[3,115] AT %IB."KUKA4_KRC4_ProfiNet_5_0".Module001_8_digital_inputs_I_115;
	::InputVariables[3,116] AT %IB."KUKA4_KRC4_ProfiNet_5_0".Module001_8_digital_inputs_I_116;
	::InputVariables[3,117] AT %IB."KUKA4_KRC4_ProfiNet_5_0".Module001_8_digital_inputs_I_117;
	::InputVariables[3,118] AT %IB."KUKA4_KRC4_ProfiNet_5_0".Module001_8_digital_inputs_I_118;
	::InputVariables[3,119] AT %IB."KUKA4_KRC4_ProfiNet_5_0".Module001_8_digital_inputs_I_119;
	::InputVariables[3,120] AT %IB."KUKA4_KRC4_ProfiNet_5_0".Module001_8_digital_inputs_I_120;
	::InputVariables[3,121] AT %IB."KUKA4_KRC4_ProfiNet_5_0".Module001_8_digital_inputs_I_121;
	::InputVariables[3,122] AT %IB."KUKA4_KRC4_ProfiNet_5_0".Module001_8_digital_inputs_I_122;
	::InputVariables[3,123] AT %IB."KUKA4_KRC4_ProfiNet_5_0".Module001_8_digital_inputs_I_123;
	::InputVariables[3,124] AT %IB."KUKA4_KRC4_ProfiNet_5_0".Module001_8_digital_inputs_I_124;
	::InputVariables[3,125] AT %IB."KUKA4_KRC4_ProfiNet_5_0".Module001_8_digital_inputs_I_125;
	::InputVariables[3,126] AT %IB."KUKA4_KRC4_ProfiNet_5_0".Module001_8_digital_inputs_I_126;
	::InputVariables[3,127] AT %IB."KUKA4_KRC4_ProfiNet_5_0".Module001_8_digital_inputs_I_127;
	::InputVariables[3,128] AT %IB."KUKA4_KRC4_ProfiNet_5_0".Module001_8_digital_inputs_I_128;
	::InputVariables[3,129] AT %IB."KUKA4_KRC4_ProfiNet_5_0".Module001_8_digital_inputs_I_129;
	::InputVariables[3,130] AT %IB."KUKA4_KRC4_ProfiNet_5_0".Module001_8_digital_inputs_I_130;
	::InputVariables[3,131] AT %IB."KUKA4_KRC4_ProfiNet_5_0".Module001_8_digital_inputs_I_131;
	::InputVariables[3,132] AT %IB."KUKA4_KRC4_ProfiNet_5_0".Module001_8_digital_inputs_I_132;
	::InputVariables[3,133] AT %IB."KUKA4_KRC4_ProfiNet_5_0".Module001_8_digital_inputs_I_133;
	::InputVariables[3,134] AT %IB."KUKA4_KRC4_ProfiNet_5_0".Module001_8_digital_inputs_I_134;
	::InputVariables[3,135] AT %IB."KUKA4_KRC4_ProfiNet_5_0".Module001_8_digital_inputs_I_135;
	::InputVariables[3,136] AT %IB."KUKA4_KRC4_ProfiNet_5_0".Module001_8_digital_inputs_I_136;
	::InputVariables[3,137] AT %IB."KUKA4_KRC4_ProfiNet_5_0".Module001_8_digital_inputs_I_137;
	::InputVariables[3,138] AT %IB."KUKA4_KRC4_ProfiNet_5_0".Module001_8_digital_inputs_I_138;
	::InputVariables[3,139] AT %IB."KUKA4_KRC4_ProfiNet_5_0".Module001_8_digital_inputs_I_139;
	::InputVariables[3,140] AT %IB."KUKA4_KRC4_ProfiNet_5_0".Module001_8_digital_inputs_I_140;
	::InputVariables[3,141] AT %IB."KUKA4_KRC4_ProfiNet_5_0".Module001_8_digital_inputs_I_141;
	::InputVariables[3,142] AT %IB."KUKA4_KRC4_ProfiNet_5_0".Module001_8_digital_inputs_I_142;
	::InputVariables[3,143] AT %IB."KUKA4_KRC4_ProfiNet_5_0".Module001_8_digital_inputs_I_143;
	::InputVariables[3,144] AT %IB."KUKA4_KRC4_ProfiNet_5_0".Module001_8_digital_inputs_I_144;
	::InputVariables[3,145] AT %IB."KUKA4_KRC4_ProfiNet_5_0".Module001_8_digital_inputs_I_145;
	::InputVariables[3,146] AT %IB."KUKA4_KRC4_ProfiNet_5_0".Module001_8_digital_inputs_I_146;
	::InputVariables[3,147] AT %IB."KUKA4_KRC4_ProfiNet_5_0".Module001_8_digital_inputs_I_147;
	::InputVariables[3,148] AT %IB."KUKA4_KRC4_ProfiNet_5_0".Module001_8_digital_inputs_I_148;
	::InputVariables[3,149] AT %IB."KUKA4_KRC4_ProfiNet_5_0".Module001_8_digital_inputs_I_149;
	::InputVariables[3,150] AT %IB."KUKA4_KRC4_ProfiNet_5_0".Module001_8_digital_inputs_I_150;
	::InputVariables[3,151] AT %IB."KUKA4_KRC4_ProfiNet_5_0".Module001_8_digital_inputs_I_151;
	::InputVariables[3,152] AT %IB."KUKA4_KRC4_ProfiNet_5_0".Module001_8_digital_inputs_I_152;
	::InputVariables[3,153] AT %IB."KUKA4_KRC4_ProfiNet_5_0".Module001_8_digital_inputs_I_153;
	::InputVariables[3,154] AT %IB."KUKA4_KRC4_ProfiNet_5_0".Module001_8_digital_inputs_I_154;
	::InputVariables[3,155] AT %IB."KUKA4_KRC4_ProfiNet_5_0".Module001_8_digital_inputs_I_155;
	::InputVariables[3,156] AT %IB."KUKA4_KRC4_ProfiNet_5_0".Module001_8_digital_inputs_I_156;
	::InputVariables[3,157] AT %IB."KUKA4_KRC4_ProfiNet_5_0".Module001_8_digital_inputs_I_157;
	::InputVariables[3,158] AT %IB."KUKA4_KRC4_ProfiNet_5_0".Module001_8_digital_inputs_I_158;
	::InputVariables[3,159] AT %IB."KUKA4_KRC4_ProfiNet_5_0".Module001_8_digital_inputs_I_159;
	::InputVariables[3,160] AT %IB."KUKA4_KRC4_ProfiNet_5_0".Module001_8_digital_inputs_I_160;
	::InputVariables[3,161] AT %IB."KUKA4_KRC4_ProfiNet_5_0".Module001_8_digital_inputs_I_161;
	::InputVariables[3,162] AT %IB."KUKA4_KRC4_ProfiNet_5_0".Module001_8_digital_inputs_I_162;
	::InputVariables[3,163] AT %IB."KUKA4_KRC4_ProfiNet_5_0".Module001_8_digital_inputs_I_163;
	::InputVariables[3,164] AT %IB."KUKA4_KRC4_ProfiNet_5_0".Module001_8_digital_inputs_I_164;
	::InputVariables[3,165] AT %IB."KUKA4_KRC4_ProfiNet_5_0".Module001_8_digital_inputs_I_165;
	::InputVariables[3,166] AT %IB."KUKA4_KRC4_ProfiNet_5_0".Module001_8_digital_inputs_I_166;
	::InputVariables[3,167] AT %IB."KUKA4_KRC4_ProfiNet_5_0".Module001_8_digital_inputs_I_167;
	::InputVariables[3,168] AT %IB."KUKA4_KRC4_ProfiNet_5_0".Module001_8_digital_inputs_I_168;
	::InputVariables[3,169] AT %IB."KUKA4_KRC4_ProfiNet_5_0".Module001_8_digital_inputs_I_169;
	::InputVariables[3,170] AT %IB."KUKA4_KRC4_ProfiNet_5_0".Module001_8_digital_inputs_I_170;
	::InputVariables[3,171] AT %IB."KUKA4_KRC4_ProfiNet_5_0".Module001_8_digital_inputs_I_171;
	::InputVariables[3,172] AT %IB."KUKA4_KRC4_ProfiNet_5_0".Module001_8_digital_inputs_I_172;
	::InputVariables[3,173] AT %IB."KUKA4_KRC4_ProfiNet_5_0".Module001_8_digital_inputs_I_173;
	::InputVariables[3,174] AT %IB."KUKA4_KRC4_ProfiNet_5_0".Module001_8_digital_inputs_I_174;
	::InputVariables[3,175] AT %IB."KUKA4_KRC4_ProfiNet_5_0".Module001_8_digital_inputs_I_175;
	::InputVariables[3,176] AT %IB."KUKA4_KRC4_ProfiNet_5_0".Module001_8_digital_inputs_I_176;
	::InputVariables[3,177] AT %IB."KUKA4_KRC4_ProfiNet_5_0".Module001_8_digital_inputs_I_177;
	::InputVariables[3,178] AT %IB."KUKA4_KRC4_ProfiNet_5_0".Module001_8_digital_inputs_I_178;
	::InputVariables[3,179] AT %IB."KUKA4_KRC4_ProfiNet_5_0".Module001_8_digital_inputs_I_179;
	::InputVariables[3,180] AT %IB."KUKA4_KRC4_ProfiNet_5_0".Module001_8_digital_inputs_I_180;
	::InputVariables[3,181] AT %IB."KUKA4_KRC4_ProfiNet_5_0".Module001_8_digital_inputs_I_181;
	::InputVariables[3,182] AT %IB."KUKA4_KRC4_ProfiNet_5_0".Module001_8_digital_inputs_I_182;
	::InputVariables[3,183] AT %IB."KUKA4_KRC4_ProfiNet_5_0".Module001_8_digital_inputs_I_183;
	::InputVariables[3,184] AT %IB."KUKA4_KRC4_ProfiNet_5_0".Module001_8_digital_inputs_I_184;
	::InputVariables[3,185] AT %IB."KUKA4_KRC4_ProfiNet_5_0".Module001_8_digital_inputs_I_185;
	::InputVariables[3,186] AT %IB."KUKA4_KRC4_ProfiNet_5_0".Module001_8_digital_inputs_I_186;
	::InputVariables[3,187] AT %IB."KUKA4_KRC4_ProfiNet_5_0".Module001_8_digital_inputs_I_187;
	::InputVariables[3,188] AT %IB."KUKA4_KRC4_ProfiNet_5_0".Module001_8_digital_inputs_I_188;
	::InputVariables[3,189] AT %IB."KUKA4_KRC4_ProfiNet_5_0".Module001_8_digital_inputs_I_189;
	::InputVariables[3,190] AT %IB."KUKA4_KRC4_ProfiNet_5_0".Module001_8_digital_inputs_I_190;
	::InputVariables[3,191] AT %IB."KUKA4_KRC4_ProfiNet_5_0".Module001_8_digital_inputs_I_191;
	::InputVariables[3,192] AT %IB."KUKA4_KRC4_ProfiNet_5_0".Module001_8_digital_inputs_I_192;
	::InputVariables[3,193] AT %IB."KUKA4_KRC4_ProfiNet_5_0".Module001_8_digital_inputs_I_193;
	::InputVariables[3,194] AT %IB."KUKA4_KRC4_ProfiNet_5_0".Module001_8_digital_inputs_I_194;
	::InputVariables[3,195] AT %IB."KUKA4_KRC4_ProfiNet_5_0".Module001_8_digital_inputs_I_195;
	::InputVariables[3,196] AT %IB."KUKA4_KRC4_ProfiNet_5_0".Module001_8_digital_inputs_I_196;
	::InputVariables[3,197] AT %IB."KUKA4_KRC4_ProfiNet_5_0".Module001_8_digital_inputs_I_197;
	::InputVariables[3,198] AT %IB."KUKA4_KRC4_ProfiNet_5_0".Module001_8_digital_inputs_I_198;
	::InputVariables[3,199] AT %IB."KUKA4_KRC4_ProfiNet_5_0".Module001_8_digital_inputs_I_199;
	::InputVariables[3,200] AT %IB."KUKA4_KRC4_ProfiNet_5_0".Module001_8_digital_inputs_I_200;
	::InputVariables[3,201] AT %IB."KUKA4_KRC4_ProfiNet_5_0".Module001_8_digital_inputs_I_201;
	::InputVariables[3,202] AT %IB."KUKA4_KRC4_ProfiNet_5_0".Module001_8_digital_inputs_I_202;
	::InputVariables[3,203] AT %IB."KUKA4_KRC4_ProfiNet_5_0".Module001_8_digital_inputs_I_203;
	::InputVariables[3,204] AT %IB."KUKA4_KRC4_ProfiNet_5_0".Module001_8_digital_inputs_I_204;
	::InputVariables[3,205] AT %IB."KUKA4_KRC4_ProfiNet_5_0".Module001_8_digital_inputs_I_205;
	::InputVariables[3,206] AT %IB."KUKA4_KRC4_ProfiNet_5_0".Module001_8_digital_inputs_I_206;
	::InputVariables[3,207] AT %IB."KUKA4_KRC4_ProfiNet_5_0".Module001_8_digital_inputs_I_207;
	::InputVariables[3,208] AT %IB."KUKA4_KRC4_ProfiNet_5_0".Module001_8_digital_inputs_I_208;
	::InputVariables[3,209] AT %IB."KUKA4_KRC4_ProfiNet_5_0".Module001_8_digital_inputs_I_209;
	::InputVariables[3,210] AT %IB."KUKA4_KRC4_ProfiNet_5_0".Module001_8_digital_inputs_I_210;
	::InputVariables[3,211] AT %IB."KUKA4_KRC4_ProfiNet_5_0".Module001_8_digital_inputs_I_211;
	::InputVariables[3,212] AT %IB."KUKA4_KRC4_ProfiNet_5_0".Module001_8_digital_inputs_I_212;
	::InputVariables[3,213] AT %IB."KUKA4_KRC4_ProfiNet_5_0".Module001_8_digital_inputs_I_213;
	::InputVariables[3,214] AT %IB."KUKA4_KRC4_ProfiNet_5_0".Module001_8_digital_inputs_I_214;
	::InputVariables[3,215] AT %IB."KUKA4_KRC4_ProfiNet_5_0".Module001_8_digital_inputs_I_215;
	::InputVariables[3,216] AT %IB."KUKA4_KRC4_ProfiNet_5_0".Module001_8_digital_inputs_I_216;
	::InputVariables[3,217] AT %IB."KUKA4_KRC4_ProfiNet_5_0".Module001_8_digital_inputs_I_217;
	::InputVariables[3,218] AT %IB."KUKA4_KRC4_ProfiNet_5_0".Module001_8_digital_inputs_I_218;
	::InputVariables[3,219] AT %IB."KUKA4_KRC4_ProfiNet_5_0".Module001_8_digital_inputs_I_219;
	::InputVariables[3,220] AT %IB."KUKA4_KRC4_ProfiNet_5_0".Module001_8_digital_inputs_I_220;
	::InputVariables[3,221] AT %IB."KUKA4_KRC4_ProfiNet_5_0".Module001_8_digital_inputs_I_221;
	::InputVariables[3,222] AT %IB."KUKA4_KRC4_ProfiNet_5_0".Module001_8_digital_inputs_I_222;
	::InputVariables[3,223] AT %IB."KUKA4_KRC4_ProfiNet_5_0".Module001_8_digital_inputs_I_223;
	::InputVariables[3,224] AT %IB."KUKA4_KRC4_ProfiNet_5_0".Module001_8_digital_inputs_I_224;
	::InputVariables[3,225] AT %IB."KUKA4_KRC4_ProfiNet_5_0".Module001_8_digital_inputs_I_225;
	::InputVariables[3,226] AT %IB."KUKA4_KRC4_ProfiNet_5_0".Module001_8_digital_inputs_I_226;
	::InputVariables[3,227] AT %IB."KUKA4_KRC4_ProfiNet_5_0".Module001_8_digital_inputs_I_227;
	::InputVariables[3,228] AT %IB."KUKA4_KRC4_ProfiNet_5_0".Module001_8_digital_inputs_I_228;
	::InputVariables[3,229] AT %IB."KUKA4_KRC4_ProfiNet_5_0".Module001_8_digital_inputs_I_229;
	::InputVariables[3,230] AT %IB."KUKA4_KRC4_ProfiNet_5_0".Module001_8_digital_inputs_I_230;
	::InputVariables[3,231] AT %IB."KUKA4_KRC4_ProfiNet_5_0".Module001_8_digital_inputs_I_231;
	::InputVariables[3,232] AT %IB."KUKA4_KRC4_ProfiNet_5_0".Module001_8_digital_inputs_I_232;
	::InputVariables[3,233] AT %IB."KUKA4_KRC4_ProfiNet_5_0".Module001_8_digital_inputs_I_233;
	::InputVariables[3,234] AT %IB."KUKA4_KRC4_ProfiNet_5_0".Module001_8_digital_inputs_I_234;
	::InputVariables[3,235] AT %IB."KUKA4_KRC4_ProfiNet_5_0".Module001_8_digital_inputs_I_235;
	::InputVariables[3,236] AT %IB."KUKA4_KRC4_ProfiNet_5_0".Module001_8_digital_inputs_I_236;
	::InputVariables[3,237] AT %IB."KUKA4_KRC4_ProfiNet_5_0".Module001_8_digital_inputs_I_237;
	::InputVariables[3,238] AT %IB."KUKA4_KRC4_ProfiNet_5_0".Module001_8_digital_inputs_I_238;
	::InputVariables[3,239] AT %IB."KUKA4_KRC4_ProfiNet_5_0".Module001_8_digital_inputs_I_239;
	::InputVariables[3,240] AT %IB."KUKA4_KRC4_ProfiNet_5_0".Module001_8_digital_inputs_I_240;
	::InputVariables[3,241] AT %IB."KUKA4_KRC4_ProfiNet_5_0".Module001_8_digital_inputs_I_241;
	::InputVariables[3,242] AT %IB."KUKA4_KRC4_ProfiNet_5_0".Module001_8_digital_inputs_I_242;
	::InputVariables[3,243] AT %IB."KUKA4_KRC4_ProfiNet_5_0".Module001_8_digital_inputs_I_243;
	::InputVariables[3,244] AT %IB."KUKA4_KRC4_ProfiNet_5_0".Module001_8_digital_inputs_I_244;
	::InputVariables[3,245] AT %IB."KUKA4_KRC4_ProfiNet_5_0".Module001_8_digital_inputs_I_245;
	::InputVariables[3,246] AT %IB."KUKA4_KRC4_ProfiNet_5_0".Module001_8_digital_inputs_I_246;
	::InputVariables[3,247] AT %IB."KUKA4_KRC4_ProfiNet_5_0".Module001_8_digital_inputs_I_247;
	::InputVariables[3,248] AT %IB."KUKA4_KRC4_ProfiNet_5_0".Module001_8_digital_inputs_I_248;
	::InputVariables[3,249] AT %IB."KUKA4_KRC4_ProfiNet_5_0".Module001_8_digital_inputs_I_249;
	::InputVariables[3,250] AT %IB."KUKA4_KRC4_ProfiNet_5_0".Module001_8_digital_inputs_I_250;
	::InputVariables[3,251] AT %IB."KUKA4_KRC4_ProfiNet_5_0".Module001_8_digital_inputs_I_251;
	::InputVariables[3,252] AT %IB."KUKA4_KRC4_ProfiNet_5_0".Module001_8_digital_inputs_I_252;
	::InputVariables[3,253] AT %IB."KUKA4_KRC4_ProfiNet_5_0".Module001_8_digital_inputs_I_253;

	::OutputVariables[3,0]	AT %QB."KUKA4_KRC4_ProfiNet_5_0".Module001_8_digital_outputs_O_00;
	::OutputVariables[3,1]	AT %QB."KUKA4_KRC4_ProfiNet_5_0".Module001_8_digital_outputs_O_01;
	::OutputVariables[3,2]	AT %QB."KUKA4_KRC4_ProfiNet_5_0".Module001_8_digital_outputs_O_02;
	::OutputVariables[3,3]	AT %QB."KUKA4_KRC4_ProfiNet_5_0".Module001_8_digital_outputs_O_03;
	::OutputVariables[3,4]	AT %QB."KUKA4_KRC4_ProfiNet_5_0".Module001_8_digital_outputs_O_04;
	::OutputVariables[3,5]	AT %QB."KUKA4_KRC4_ProfiNet_5_0".Module001_8_digital_outputs_O_05;
	::OutputVariables[3,6]	AT %QB."KUKA4_KRC4_ProfiNet_5_0".Module001_8_digital_outputs_O_06;
	::OutputVariables[3,7]	AT %QB."KUKA4_KRC4_ProfiNet_5_0".Module001_8_digital_outputs_O_07;
	::OutputVariables[3,8]	AT %QB."KUKA4_KRC4_ProfiNet_5_0".Module001_8_digital_outputs_O_08;
	::OutputVariables[3,9]	AT %QB."KUKA4_KRC4_ProfiNet_5_0".Module001_8_digital_outputs_O_09;
	::OutputVariables[3,10]	AT %QB."KUKA4_KRC4_ProfiNet_5_0".Module001_8_digital_outputs_O_10;
	::OutputVariables[3,11]	AT %QB."KUKA4_KRC4_ProfiNet_5_0".Module001_8_digital_outputs_O_11;
	::OutputVariables[3,12]	AT %QB."KUKA4_KRC4_ProfiNet_5_0".Module001_8_digital_outputs_O_12;
	::OutputVariables[3,13]	AT %QB."KUKA4_KRC4_ProfiNet_5_0".Module001_8_digital_outputs_O_13;
	::OutputVariables[3,14]	AT %QB."KUKA4_KRC4_ProfiNet_5_0".Module001_8_digital_outputs_O_14;
	::OutputVariables[3,15]	AT %QB."KUKA4_KRC4_ProfiNet_5_0".Module001_8_digital_outputs_O_15;
	::OutputVariables[3,16]	AT %QB."KUKA4_KRC4_ProfiNet_5_0".Module001_8_digital_outputs_O_16;
	::OutputVariables[3,17]	AT %QB."KUKA4_KRC4_ProfiNet_5_0".Module001_8_digital_outputs_O_17;
	::OutputVariables[3,18]	AT %QB."KUKA4_KRC4_ProfiNet_5_0".Module001_8_digital_outputs_O_18;
	::OutputVariables[3,19]	AT %QB."KUKA4_KRC4_ProfiNet_5_0".Module001_8_digital_outputs_O_19;
	::OutputVariables[3,20]	AT %QB."KUKA4_KRC4_ProfiNet_5_0".Module001_8_digital_outputs_O_20;
	::OutputVariables[3,21]	AT %QB."KUKA4_KRC4_ProfiNet_5_0".Module001_8_digital_outputs_O_21;
	::OutputVariables[3,22]	AT %QB."KUKA4_KRC4_ProfiNet_5_0".Module001_8_digital_outputs_O_22;
	::OutputVariables[3,23]	AT %QB."KUKA4_KRC4_ProfiNet_5_0".Module001_8_digital_outputs_O_23;
	::OutputVariables[3,24]	AT %QB."KUKA4_KRC4_ProfiNet_5_0".Module001_8_digital_outputs_O_24;
	::OutputVariables[3,25]	AT %QB."KUKA4_KRC4_ProfiNet_5_0".Module001_8_digital_outputs_O_25;
	::OutputVariables[3,26]	AT %QB."KUKA4_KRC4_ProfiNet_5_0".Module001_8_digital_outputs_O_26;
	::OutputVariables[3,27]	AT %QB."KUKA4_KRC4_ProfiNet_5_0".Module001_8_digital_outputs_O_27;
	::OutputVariables[3,28]	AT %QB."KUKA4_KRC4_ProfiNet_5_0".Module001_8_digital_outputs_O_28;
	::OutputVariables[3,29]	AT %QB."KUKA4_KRC4_ProfiNet_5_0".Module001_8_digital_outputs_O_29;
	::OutputVariables[3,30]	AT %QB."KUKA4_KRC4_ProfiNet_5_0".Module001_8_digital_outputs_O_30;
	::OutputVariables[3,31]	AT %QB."KUKA4_KRC4_ProfiNet_5_0".Module001_8_digital_outputs_O_31;
	::OutputVariables[3,32]	AT %QB."KUKA4_KRC4_ProfiNet_5_0".Module001_8_digital_outputs_O_32;
	::OutputVariables[3,33]	AT %QB."KUKA4_KRC4_ProfiNet_5_0".Module001_8_digital_outputs_O_33;
	::OutputVariables[3,34]	AT %QB."KUKA4_KRC4_ProfiNet_5_0".Module001_8_digital_outputs_O_34;
	::OutputVariables[3,35]	AT %QB."KUKA4_KRC4_ProfiNet_5_0".Module001_8_digital_outputs_O_35;
	::OutputVariables[3,36]	AT %QB."KUKA4_KRC4_ProfiNet_5_0".Module001_8_digital_outputs_O_36;
	::OutputVariables[3,37]	AT %QB."KUKA4_KRC4_ProfiNet_5_0".Module001_8_digital_outputs_O_37;
	::OutputVariables[3,38]	AT %QB."KUKA4_KRC4_ProfiNet_5_0".Module001_8_digital_outputs_O_38;
	::OutputVariables[3,39]	AT %QB."KUKA4_KRC4_ProfiNet_5_0".Module001_8_digital_outputs_O_39;
	::OutputVariables[3,40]	AT %QB."KUKA4_KRC4_ProfiNet_5_0".Module001_8_digital_outputs_O_40;
	::OutputVariables[3,41]	AT %QB."KUKA4_KRC4_ProfiNet_5_0".Module001_8_digital_outputs_O_41;
	::OutputVariables[3,42]	AT %QB."KUKA4_KRC4_ProfiNet_5_0".Module001_8_digital_outputs_O_42;
	::OutputVariables[3,43]	AT %QB."KUKA4_KRC4_ProfiNet_5_0".Module001_8_digital_outputs_O_43;
	::OutputVariables[3,44]	AT %QB."KUKA4_KRC4_ProfiNet_5_0".Module001_8_digital_outputs_O_44;
	::OutputVariables[3,45]	AT %QB."KUKA4_KRC4_ProfiNet_5_0".Module001_8_digital_outputs_O_45;
	::OutputVariables[3,46]	AT %QB."KUKA4_KRC4_ProfiNet_5_0".Module001_8_digital_outputs_O_46;
	::OutputVariables[3,47]	AT %QB."KUKA4_KRC4_ProfiNet_5_0".Module001_8_digital_outputs_O_47;
	::OutputVariables[3,48]	AT %QB."KUKA4_KRC4_ProfiNet_5_0".Module001_8_digital_outputs_O_48;
	::OutputVariables[3,49]	AT %QB."KUKA4_KRC4_ProfiNet_5_0".Module001_8_digital_outputs_O_49;
	::OutputVariables[3,50]	AT %QB."KUKA4_KRC4_ProfiNet_5_0".Module001_8_digital_outputs_O_50;
	::OutputVariables[3,51]	AT %QB."KUKA4_KRC4_ProfiNet_5_0".Module001_8_digital_outputs_O_51;
	::OutputVariables[3,52]	AT %QB."KUKA4_KRC4_ProfiNet_5_0".Module001_8_digital_outputs_O_52;
	::OutputVariables[3,53]	AT %QB."KUKA4_KRC4_ProfiNet_5_0".Module001_8_digital_outputs_O_53;
	::OutputVariables[3,54]	AT %QB."KUKA4_KRC4_ProfiNet_5_0".Module001_8_digital_outputs_O_54;
	::OutputVariables[3,55]	AT %QB."KUKA4_KRC4_ProfiNet_5_0".Module001_8_digital_outputs_O_55;
	::OutputVariables[3,56]	AT %QB."KUKA4_KRC4_ProfiNet_5_0".Module001_8_digital_outputs_O_56;
	::OutputVariables[3,57]	AT %QB."KUKA4_KRC4_ProfiNet_5_0".Module001_8_digital_outputs_O_57;
	::OutputVariables[3,58]	AT %QB."KUKA4_KRC4_ProfiNet_5_0".Module001_8_digital_outputs_O_58;
	::OutputVariables[3,59]	AT %QB."KUKA4_KRC4_ProfiNet_5_0".Module001_8_digital_outputs_O_59;
	::OutputVariables[3,60]	AT %QB."KUKA4_KRC4_ProfiNet_5_0".Module001_8_digital_outputs_O_60;
	::OutputVariables[3,61]	AT %QB."KUKA4_KRC4_ProfiNet_5_0".Module001_8_digital_outputs_O_61;
	::OutputVariables[3,62]	AT %QB."KUKA4_KRC4_ProfiNet_5_0".Module001_8_digital_outputs_O_62;
	::OutputVariables[3,63]	AT %QB."KUKA4_KRC4_ProfiNet_5_0".Module001_8_digital_outputs_O_63;
	::OutputVariables[3,64]	AT %QB."KUKA4_KRC4_ProfiNet_5_0".Module001_8_digital_outputs_O_64;
	::OutputVariables[3,65]	AT %QB."KUKA4_KRC4_ProfiNet_5_0".Module001_8_digital_outputs_O_65;
	::OutputVariables[3,66]	AT %QB."KUKA4_KRC4_ProfiNet_5_0".Module001_8_digital_outputs_O_66;
	::OutputVariables[3,67]	AT %QB."KUKA4_KRC4_ProfiNet_5_0".Module001_8_digital_outputs_O_67;
	::OutputVariables[3,68]	AT %QB."KUKA4_KRC4_ProfiNet_5_0".Module001_8_digital_outputs_O_68;
	::OutputVariables[3,69]	AT %QB."KUKA4_KRC4_ProfiNet_5_0".Module001_8_digital_outputs_O_69;
	::OutputVariables[3,70]	AT %QB."KUKA4_KRC4_ProfiNet_5_0".Module001_8_digital_outputs_O_70;
	::OutputVariables[3,71]	AT %QB."KUKA4_KRC4_ProfiNet_5_0".Module001_8_digital_outputs_O_71;
	::OutputVariables[3,72]	AT %QB."KUKA4_KRC4_ProfiNet_5_0".Module001_8_digital_outputs_O_72;
	::OutputVariables[3,73]	AT %QB."KUKA4_KRC4_ProfiNet_5_0".Module001_8_digital_outputs_O_73;
	::OutputVariables[3,74]	AT %QB."KUKA4_KRC4_ProfiNet_5_0".Module001_8_digital_outputs_O_74;
	::OutputVariables[3,75]	AT %QB."KUKA4_KRC4_ProfiNet_5_0".Module001_8_digital_outputs_O_75;
	::OutputVariables[3,76]	AT %QB."KUKA4_KRC4_ProfiNet_5_0".Module001_8_digital_outputs_O_76;
	::OutputVariables[3,77]	AT %QB."KUKA4_KRC4_ProfiNet_5_0".Module001_8_digital_outputs_O_77;
	::OutputVariables[3,78]	AT %QB."KUKA4_KRC4_ProfiNet_5_0".Module001_8_digital_outputs_O_78;
	::OutputVariables[3,79]	AT %QB."KUKA4_KRC4_ProfiNet_5_0".Module001_8_digital_outputs_O_79;
	::OutputVariables[3,80]	AT %QB."KUKA4_KRC4_ProfiNet_5_0".Module001_8_digital_outputs_O_80;
	::OutputVariables[3,81]	AT %QB."KUKA4_KRC4_ProfiNet_5_0".Module001_8_digital_outputs_O_81;
	::OutputVariables[3,82]	AT %QB."KUKA4_KRC4_ProfiNet_5_0".Module001_8_digital_outputs_O_82;
	::OutputVariables[3,83]	AT %QB."KUKA4_KRC4_ProfiNet_5_0".Module001_8_digital_outputs_O_83;
	::OutputVariables[3,84]	AT %QB."KUKA4_KRC4_ProfiNet_5_0".Module001_8_digital_outputs_O_84;
	::OutputVariables[3,85]	AT %QB."KUKA4_KRC4_ProfiNet_5_0".Module001_8_digital_outputs_O_85;
	::OutputVariables[3,86]	AT %QB."KUKA4_KRC4_ProfiNet_5_0".Module001_8_digital_outputs_O_86;
	::OutputVariables[3,87]	AT %QB."KUKA4_KRC4_ProfiNet_5_0".Module001_8_digital_outputs_O_87;
	::OutputVariables[3,88]	AT %QB."KUKA4_KRC4_ProfiNet_5_0".Module001_8_digital_outputs_O_88;
	::OutputVariables[3,89]	AT %QB."KUKA4_KRC4_ProfiNet_5_0".Module001_8_digital_outputs_O_89;
	::OutputVariables[3,90]	AT %QB."KUKA4_KRC4_ProfiNet_5_0".Module001_8_digital_outputs_O_90;
	::OutputVariables[3,91]	AT %QB."KUKA4_KRC4_ProfiNet_5_0".Module001_8_digital_outputs_O_91;
	::OutputVariables[3,92]	AT %QB."KUKA4_KRC4_ProfiNet_5_0".Module001_8_digital_outputs_O_92;
	::OutputVariables[3,93]	AT %QB."KUKA4_KRC4_ProfiNet_5_0".Module001_8_digital_outputs_O_93;
	::OutputVariables[3,94]	AT %QB."KUKA4_KRC4_ProfiNet_5_0".Module001_8_digital_outputs_O_94;
	::OutputVariables[3,95]	AT %QB."KUKA4_KRC4_ProfiNet_5_0".Module001_8_digital_outputs_O_95;
	::OutputVariables[3,96]	AT %QB."KUKA4_KRC4_ProfiNet_5_0".Module001_8_digital_outputs_O_96;
	::OutputVariables[3,97]	AT %QB."KUKA4_KRC4_ProfiNet_5_0".Module001_8_digital_outputs_O_97;
	::OutputVariables[3,98]	AT %QB."KUKA4_KRC4_ProfiNet_5_0".Module001_8_digital_outputs_O_98;
	::OutputVariables[3,99]	AT %QB."KUKA4_KRC4_ProfiNet_5_0".Module001_8_digital_outputs_O_99;
	::OutputVariables[3,100]	AT %QB."KUKA4_KRC4_ProfiNet_5_0".Module001_8_digital_outputs_O_100;
	::OutputVariables[3,101]	AT %QB."KUKA4_KRC4_ProfiNet_5_0".Module001_8_digital_outputs_O_101;
	::OutputVariables[3,102]	AT %QB."KUKA4_KRC4_ProfiNet_5_0".Module001_8_digital_outputs_O_102;
	::OutputVariables[3,103]	AT %QB."KUKA4_KRC4_ProfiNet_5_0".Module001_8_digital_outputs_O_103;
	::OutputVariables[3,104]	AT %QB."KUKA4_KRC4_ProfiNet_5_0".Module001_8_digital_outputs_O_104;
	::OutputVariables[3,105]	AT %QB."KUKA4_KRC4_ProfiNet_5_0".Module001_8_digital_outputs_O_105;
	::OutputVariables[3,106]	AT %QB."KUKA4_KRC4_ProfiNet_5_0".Module001_8_digital_outputs_O_106;
	::OutputVariables[3,107]	AT %QB."KUKA4_KRC4_ProfiNet_5_0".Module001_8_digital_outputs_O_107;
	::OutputVariables[3,108]	AT %QB."KUKA4_KRC4_ProfiNet_5_0".Module001_8_digital_outputs_O_108;
	::OutputVariables[3,109]	AT %QB."KUKA4_KRC4_ProfiNet_5_0".Module001_8_digital_outputs_O_109;
	::OutputVariables[3,110]	AT %QB."KUKA4_KRC4_ProfiNet_5_0".Module001_8_digital_outputs_O_110;
	::OutputVariables[3,111]	AT %QB."KUKA4_KRC4_ProfiNet_5_0".Module001_8_digital_outputs_O_111;
	::OutputVariables[3,112]	AT %QB."KUKA4_KRC4_ProfiNet_5_0".Module001_8_digital_outputs_O_112;
	::OutputVariables[3,113]	AT %QB."KUKA4_KRC4_ProfiNet_5_0".Module001_8_digital_outputs_O_113;
	::OutputVariables[3,114]	AT %QB."KUKA4_KRC4_ProfiNet_5_0".Module001_8_digital_outputs_O_114;
	::OutputVariables[3,115]	AT %QB."KUKA4_KRC4_ProfiNet_5_0".Module001_8_digital_outputs_O_115;
	::OutputVariables[3,116]	AT %QB."KUKA4_KRC4_ProfiNet_5_0".Module001_8_digital_outputs_O_116;
	::OutputVariables[3,117]	AT %QB."KUKA4_KRC4_ProfiNet_5_0".Module001_8_digital_outputs_O_117;
	::OutputVariables[3,118]	AT %QB."KUKA4_KRC4_ProfiNet_5_0".Module001_8_digital_outputs_O_118;
	::OutputVariables[3,119]	AT %QB."KUKA4_KRC4_ProfiNet_5_0".Module001_8_digital_outputs_O_119;
	::OutputVariables[3,120]	AT %QB."KUKA4_KRC4_ProfiNet_5_0".Module001_8_digital_outputs_O_120;
	::OutputVariables[3,121]	AT %QB."KUKA4_KRC4_ProfiNet_5_0".Module001_8_digital_outputs_O_121;
	::OutputVariables[3,122]	AT %QB."KUKA4_KRC4_ProfiNet_5_0".Module001_8_digital_outputs_O_122;
	::OutputVariables[3,123]	AT %QB."KUKA4_KRC4_ProfiNet_5_0".Module001_8_digital_outputs_O_123;
	::OutputVariables[3,124]	AT %QB."KUKA4_KRC4_ProfiNet_5_0".Module001_8_digital_outputs_O_124;
	::OutputVariables[3,125]	AT %QB."KUKA4_KRC4_ProfiNet_5_0".Module001_8_digital_outputs_O_125;
	::OutputVariables[3,126]	AT %QB."KUKA4_KRC4_ProfiNet_5_0".Module001_8_digital_outputs_O_126;
	::OutputVariables[3,127]	AT %QB."KUKA4_KRC4_ProfiNet_5_0".Module001_8_digital_outputs_O_127;
	::OutputVariables[3,128]	AT %QB."KUKA4_KRC4_ProfiNet_5_0".Module001_8_digital_outputs_O_128;
	::OutputVariables[3,129]	AT %QB."KUKA4_KRC4_ProfiNet_5_0".Module001_8_digital_outputs_O_129;
	::OutputVariables[3,130]	AT %QB."KUKA4_KRC4_ProfiNet_5_0".Module001_8_digital_outputs_O_130;
	::OutputVariables[3,131]	AT %QB."KUKA4_KRC4_ProfiNet_5_0".Module001_8_digital_outputs_O_131;
	::OutputVariables[3,132]	AT %QB."KUKA4_KRC4_ProfiNet_5_0".Module001_8_digital_outputs_O_132;
	::OutputVariables[3,133]	AT %QB."KUKA4_KRC4_ProfiNet_5_0".Module001_8_digital_outputs_O_133;
	::OutputVariables[3,134]	AT %QB."KUKA4_KRC4_ProfiNet_5_0".Module001_8_digital_outputs_O_134;
	::OutputVariables[3,135]	AT %QB."KUKA4_KRC4_ProfiNet_5_0".Module001_8_digital_outputs_O_135;
	::OutputVariables[3,136]	AT %QB."KUKA4_KRC4_ProfiNet_5_0".Module001_8_digital_outputs_O_136;
	::OutputVariables[3,137]	AT %QB."KUKA4_KRC4_ProfiNet_5_0".Module001_8_digital_outputs_O_137;
	::OutputVariables[3,138]	AT %QB."KUKA4_KRC4_ProfiNet_5_0".Module001_8_digital_outputs_O_138;
	::OutputVariables[3,139]	AT %QB."KUKA4_KRC4_ProfiNet_5_0".Module001_8_digital_outputs_O_139;
	::OutputVariables[3,140]	AT %QB."KUKA4_KRC4_ProfiNet_5_0".Module001_8_digital_outputs_O_140;
	::OutputVariables[3,141]	AT %QB."KUKA4_KRC4_ProfiNet_5_0".Module001_8_digital_outputs_O_141;
	::OutputVariables[3,142]	AT %QB."KUKA4_KRC4_ProfiNet_5_0".Module001_8_digital_outputs_O_142;
	::OutputVariables[3,143]	AT %QB."KUKA4_KRC4_ProfiNet_5_0".Module001_8_digital_outputs_O_143;
	::OutputVariables[3,144]	AT %QB."KUKA4_KRC4_ProfiNet_5_0".Module001_8_digital_outputs_O_144;
	::OutputVariables[3,145]	AT %QB."KUKA4_KRC4_ProfiNet_5_0".Module001_8_digital_outputs_O_145;
	::OutputVariables[3,146]	AT %QB."KUKA4_KRC4_ProfiNet_5_0".Module001_8_digital_outputs_O_146;
	::OutputVariables[3,147]	AT %QB."KUKA4_KRC4_ProfiNet_5_0".Module001_8_digital_outputs_O_147;
	::OutputVariables[3,148]	AT %QB."KUKA4_KRC4_ProfiNet_5_0".Module001_8_digital_outputs_O_148;
	::OutputVariables[3,149]	AT %QB."KUKA4_KRC4_ProfiNet_5_0".Module001_8_digital_outputs_O_149;
	::OutputVariables[3,150]	AT %QB."KUKA4_KRC4_ProfiNet_5_0".Module001_8_digital_outputs_O_150;
	::OutputVariables[3,151]	AT %QB."KUKA4_KRC4_ProfiNet_5_0".Module001_8_digital_outputs_O_151;
	::OutputVariables[3,152]	AT %QB."KUKA4_KRC4_ProfiNet_5_0".Module001_8_digital_outputs_O_152;
	::OutputVariables[3,153]	AT %QB."KUKA4_KRC4_ProfiNet_5_0".Module001_8_digital_outputs_O_153;
	::OutputVariables[3,154]	AT %QB."KUKA4_KRC4_ProfiNet_5_0".Module001_8_digital_outputs_O_154;
	::OutputVariables[3,155]	AT %QB."KUKA4_KRC4_ProfiNet_5_0".Module001_8_digital_outputs_O_155;
	::OutputVariables[3,156]	AT %QB."KUKA4_KRC4_ProfiNet_5_0".Module001_8_digital_outputs_O_156;
	::OutputVariables[3,157]	AT %QB."KUKA4_KRC4_ProfiNet_5_0".Module001_8_digital_outputs_O_157;
	::OutputVariables[3,158]	AT %QB."KUKA4_KRC4_ProfiNet_5_0".Module001_8_digital_outputs_O_158;
	::OutputVariables[3,159]	AT %QB."KUKA4_KRC4_ProfiNet_5_0".Module001_8_digital_outputs_O_159;
	::OutputVariables[3,160]	AT %QB."KUKA4_KRC4_ProfiNet_5_0".Module001_8_digital_outputs_O_160;
	::OutputVariables[3,161]	AT %QB."KUKA4_KRC4_ProfiNet_5_0".Module001_8_digital_outputs_O_161;
	::OutputVariables[3,162]	AT %QB."KUKA4_KRC4_ProfiNet_5_0".Module001_8_digital_outputs_O_162;
	::OutputVariables[3,163]	AT %QB."KUKA4_KRC4_ProfiNet_5_0".Module001_8_digital_outputs_O_163;
	::OutputVariables[3,164]	AT %QB."KUKA4_KRC4_ProfiNet_5_0".Module001_8_digital_outputs_O_164;
	::OutputVariables[3,165]	AT %QB."KUKA4_KRC4_ProfiNet_5_0".Module001_8_digital_outputs_O_165;
	::OutputVariables[3,166]	AT %QB."KUKA4_KRC4_ProfiNet_5_0".Module001_8_digital_outputs_O_166;
	::OutputVariables[3,167]	AT %QB."KUKA4_KRC4_ProfiNet_5_0".Module001_8_digital_outputs_O_167;
	::OutputVariables[3,168]	AT %QB."KUKA4_KRC4_ProfiNet_5_0".Module001_8_digital_outputs_O_168;
	::OutputVariables[3,169]	AT %QB."KUKA4_KRC4_ProfiNet_5_0".Module001_8_digital_outputs_O_169;
	::OutputVariables[3,170]	AT %QB."KUKA4_KRC4_ProfiNet_5_0".Module001_8_digital_outputs_O_170;
	::OutputVariables[3,171]	AT %QB."KUKA4_KRC4_ProfiNet_5_0".Module001_8_digital_outputs_O_171;
	::OutputVariables[3,172]	AT %QB."KUKA4_KRC4_ProfiNet_5_0".Module001_8_digital_outputs_O_172;
	::OutputVariables[3,173]	AT %QB."KUKA4_KRC4_ProfiNet_5_0".Module001_8_digital_outputs_O_173;
	::OutputVariables[3,174]	AT %QB."KUKA4_KRC4_ProfiNet_5_0".Module001_8_digital_outputs_O_174;
	::OutputVariables[3,175]	AT %QB."KUKA4_KRC4_ProfiNet_5_0".Module001_8_digital_outputs_O_175;
	::OutputVariables[3,176]	AT %QB."KUKA4_KRC4_ProfiNet_5_0".Module001_8_digital_outputs_O_176;
	::OutputVariables[3,177]	AT %QB."KUKA4_KRC4_ProfiNet_5_0".Module001_8_digital_outputs_O_177;
	::OutputVariables[3,178]	AT %QB."KUKA4_KRC4_ProfiNet_5_0".Module001_8_digital_outputs_O_178;
	::OutputVariables[3,179]	AT %QB."KUKA4_KRC4_ProfiNet_5_0".Module001_8_digital_outputs_O_179;
	::OutputVariables[3,180]	AT %QB."KUKA4_KRC4_ProfiNet_5_0".Module001_8_digital_outputs_O_180;
	::OutputVariables[3,181]	AT %QB."KUKA4_KRC4_ProfiNet_5_0".Module001_8_digital_outputs_O_181;
	::OutputVariables[3,182]	AT %QB."KUKA4_KRC4_ProfiNet_5_0".Module001_8_digital_outputs_O_182;
	::OutputVariables[3,183]	AT %QB."KUKA4_KRC4_ProfiNet_5_0".Module001_8_digital_outputs_O_183;
	::OutputVariables[3,184]	AT %QB."KUKA4_KRC4_ProfiNet_5_0".Module001_8_digital_outputs_O_184;
	::OutputVariables[3,185]	AT %QB."KUKA4_KRC4_ProfiNet_5_0".Module001_8_digital_outputs_O_185;
	::OutputVariables[3,186]	AT %QB."KUKA4_KRC4_ProfiNet_5_0".Module001_8_digital_outputs_O_186;
	::OutputVariables[3,187]	AT %QB."KUKA4_KRC4_ProfiNet_5_0".Module001_8_digital_outputs_O_187;
	::OutputVariables[3,188]	AT %QB."KUKA4_KRC4_ProfiNet_5_0".Module001_8_digital_outputs_O_188;
	::OutputVariables[3,189]	AT %QB."KUKA4_KRC4_ProfiNet_5_0".Module001_8_digital_outputs_O_189;
	::OutputVariables[3,190]	AT %QB."KUKA4_KRC4_ProfiNet_5_0".Module001_8_digital_outputs_O_190;
	::OutputVariables[3,191]	AT %QB."KUKA4_KRC4_ProfiNet_5_0".Module001_8_digital_outputs_O_191;
	::OutputVariables[3,192]	AT %QB."KUKA4_KRC4_ProfiNet_5_0".Module001_8_digital_outputs_O_192;
	::OutputVariables[3,193]	AT %QB."KUKA4_KRC4_ProfiNet_5_0".Module001_8_digital_outputs_O_193;
	::OutputVariables[3,194]	AT %QB."KUKA4_KRC4_ProfiNet_5_0".Module001_8_digital_outputs_O_194;
	::OutputVariables[3,195]	AT %QB."KUKA4_KRC4_ProfiNet_5_0".Module001_8_digital_outputs_O_195;
	::OutputVariables[3,196]	AT %QB."KUKA4_KRC4_ProfiNet_5_0".Module001_8_digital_outputs_O_196;
	::OutputVariables[3,197]	AT %QB."KUKA4_KRC4_ProfiNet_5_0".Module001_8_digital_outputs_O_197;
	::OutputVariables[3,198]	AT %QB."KUKA4_KRC4_ProfiNet_5_0".Module001_8_digital_outputs_O_198;
	::OutputVariables[3,199]	AT %QB."KUKA4_KRC4_ProfiNet_5_0".Module001_8_digital_outputs_O_199;
	::OutputVariables[3,200]	AT %QB."KUKA4_KRC4_ProfiNet_5_0".Module001_8_digital_outputs_O_200;
	::OutputVariables[3,201]	AT %QB."KUKA4_KRC4_ProfiNet_5_0".Module001_8_digital_outputs_O_201;
	::OutputVariables[3,202]	AT %QB."KUKA4_KRC4_ProfiNet_5_0".Module001_8_digital_outputs_O_202;
	::OutputVariables[3,203]	AT %QB."KUKA4_KRC4_ProfiNet_5_0".Module001_8_digital_outputs_O_203;
	::OutputVariables[3,204]	AT %QB."KUKA4_KRC4_ProfiNet_5_0".Module001_8_digital_outputs_O_204;
	::OutputVariables[3,205]	AT %QB."KUKA4_KRC4_ProfiNet_5_0".Module001_8_digital_outputs_O_205;
	::OutputVariables[3,206]	AT %QB."KUKA4_KRC4_ProfiNet_5_0".Module001_8_digital_outputs_O_206;
	::OutputVariables[3,207]	AT %QB."KUKA4_KRC4_ProfiNet_5_0".Module001_8_digital_outputs_O_207;
	::OutputVariables[3,208]	AT %QB."KUKA4_KRC4_ProfiNet_5_0".Module001_8_digital_outputs_O_208;
	::OutputVariables[3,209]	AT %QB."KUKA4_KRC4_ProfiNet_5_0".Module001_8_digital_outputs_O_209;
	::OutputVariables[3,210]	AT %QB."KUKA4_KRC4_ProfiNet_5_0".Module001_8_digital_outputs_O_210;
	::OutputVariables[3,211]	AT %QB."KUKA4_KRC4_ProfiNet_5_0".Module001_8_digital_outputs_O_211;
	::OutputVariables[3,212]	AT %QB."KUKA4_KRC4_ProfiNet_5_0".Module001_8_digital_outputs_O_212;
	::OutputVariables[3,213]	AT %QB."KUKA4_KRC4_ProfiNet_5_0".Module001_8_digital_outputs_O_213;
	::OutputVariables[3,214]	AT %QB."KUKA4_KRC4_ProfiNet_5_0".Module001_8_digital_outputs_O_214;
	::OutputVariables[3,215]	AT %QB."KUKA4_KRC4_ProfiNet_5_0".Module001_8_digital_outputs_O_215;
	::OutputVariables[3,216]	AT %QB."KUKA4_KRC4_ProfiNet_5_0".Module001_8_digital_outputs_O_216;
	::OutputVariables[3,217]	AT %QB."KUKA4_KRC4_ProfiNet_5_0".Module001_8_digital_outputs_O_217;
	::OutputVariables[3,218]	AT %QB."KUKA4_KRC4_ProfiNet_5_0".Module001_8_digital_outputs_O_218;
	::OutputVariables[3,219]	AT %QB."KUKA4_KRC4_ProfiNet_5_0".Module001_8_digital_outputs_O_219;
	::OutputVariables[3,220]	AT %QB."KUKA4_KRC4_ProfiNet_5_0".Module001_8_digital_outputs_O_220;
	::OutputVariables[3,221]	AT %QB."KUKA4_KRC4_ProfiNet_5_0".Module001_8_digital_outputs_O_221;
	::OutputVariables[3,222]	AT %QB."KUKA4_KRC4_ProfiNet_5_0".Module001_8_digital_outputs_O_222;
	::OutputVariables[3,223]	AT %QB."KUKA4_KRC4_ProfiNet_5_0".Module001_8_digital_outputs_O_223;
	::OutputVariables[3,224]	AT %QB."KUKA4_KRC4_ProfiNet_5_0".Module001_8_digital_outputs_O_224;
	::OutputVariables[3,225]	AT %QB."KUKA4_KRC4_ProfiNet_5_0".Module001_8_digital_outputs_O_225;
	::OutputVariables[3,226]	AT %QB."KUKA4_KRC4_ProfiNet_5_0".Module001_8_digital_outputs_O_226;
	::OutputVariables[3,227]	AT %QB."KUKA4_KRC4_ProfiNet_5_0".Module001_8_digital_outputs_O_227;
	::OutputVariables[3,228]	AT %QB."KUKA4_KRC4_ProfiNet_5_0".Module001_8_digital_outputs_O_228;
	::OutputVariables[3,229]	AT %QB."KUKA4_KRC4_ProfiNet_5_0".Module001_8_digital_outputs_O_229;
	::OutputVariables[3,230]	AT %QB."KUKA4_KRC4_ProfiNet_5_0".Module001_8_digital_outputs_O_230;
	::OutputVariables[3,231]	AT %QB."KUKA4_KRC4_ProfiNet_5_0".Module001_8_digital_outputs_O_231;
	::OutputVariables[3,232]	AT %QB."KUKA4_KRC4_ProfiNet_5_0".Module001_8_digital_outputs_O_232;
	::OutputVariables[3,233]	AT %QB."KUKA4_KRC4_ProfiNet_5_0".Module001_8_digital_outputs_O_233;
	::OutputVariables[3,234]	AT %QB."KUKA4_KRC4_ProfiNet_5_0".Module001_8_digital_outputs_O_234;
	::OutputVariables[3,235]	AT %QB."KUKA4_KRC4_ProfiNet_5_0".Module001_8_digital_outputs_O_235;
	::OutputVariables[3,236]	AT %QB."KUKA4_KRC4_ProfiNet_5_0".Module001_8_digital_outputs_O_236;
	::OutputVariables[3,237]	AT %QB."KUKA4_KRC4_ProfiNet_5_0".Module001_8_digital_outputs_O_237;
	::OutputVariables[3,238]	AT %QB."KUKA4_KRC4_ProfiNet_5_0".Module001_8_digital_outputs_O_238;
	::OutputVariables[3,239]	AT %QB."KUKA4_KRC4_ProfiNet_5_0".Module001_8_digital_outputs_O_239;
	::OutputVariables[3,240]	AT %QB."KUKA4_KRC4_ProfiNet_5_0".Module001_8_digital_outputs_O_240;
	::OutputVariables[3,241]	AT %QB."KUKA4_KRC4_ProfiNet_5_0".Module001_8_digital_outputs_O_241;
	::OutputVariables[3,242]	AT %QB."KUKA4_KRC4_ProfiNet_5_0".Module001_8_digital_outputs_O_242;
	::OutputVariables[3,243]	AT %QB."KUKA4_KRC4_ProfiNet_5_0".Module001_8_digital_outputs_O_243;
	::OutputVariables[3,244]	AT %QB."KUKA4_KRC4_ProfiNet_5_0".Module001_8_digital_outputs_O_244;
	::OutputVariables[3,245]	AT %QB."KUKA4_KRC4_ProfiNet_5_0".Module001_8_digital_outputs_O_245;
	::OutputVariables[3,246]	AT %QB."KUKA4_KRC4_ProfiNet_5_0".Module001_8_digital_outputs_O_246;
	::OutputVariables[3,247]	AT %QB."KUKA4_KRC4_ProfiNet_5_0".Module001_8_digital_outputs_O_247;
	::OutputVariables[3,248]	AT %QB."KUKA4_KRC4_ProfiNet_5_0".Module001_8_digital_outputs_O_248;
	::OutputVariables[3,249]	AT %QB."KUKA4_KRC4_ProfiNet_5_0".Module001_8_digital_outputs_O_249;
	::OutputVariables[3,250]	AT %QB."KUKA4_KRC4_ProfiNet_5_0".Module001_8_digital_outputs_O_250;
	::OutputVariables[3,251]	AT %QB."KUKA4_KRC4_ProfiNet_5_0".Module001_8_digital_outputs_O_251;
	::OutputVariables[3,252]	AT %QB."KUKA4_KRC4_ProfiNet_5_0".Module001_8_digital_outputs_O_252;
	::OutputVariables[3,253]	AT %QB."KUKA4_KRC4_ProfiNet_5_0".Module001_8_digital_outputs_O_253;
```
